LIN {X 0,Y 351.6,Z 693.303,A -85,B 0,C 180,E1 16687.079,E2 16687.079} C_VEL
LIN {X 0,Y 338.557,Z 672.287,A -85,B 0,C 180,E1 16684.342,E2 16684.342} C_VEL
LIN {X 0,Y 333.384,Z 663.984,A -85,B 0,C 180,E1 16683.188,E2 16683.188} C_VEL
LIN {X 0,Y 331.512,Z 660.817,A -85,B 0,C 180,E1 16682.749,E2 16682.749} C_VEL
LIN {X 0,Y 331.209,Z 659.403,A -85,B 0,C 180,E1 16682.628,E2 16682.628} C_VEL
LIN {X 0,Y 331.206,Z 659.412,A -85,B 0,C 180,E1 16678.295,E2 16678.295} C_VEL
LIN {X 0,Y 331.179,Z 659.421,A -85,B 0,C 180,E1 16674.056,E2 16674.056} C_VEL
LIN {X 0,Y 331.185,Z 659.414,A -85,B 0,C 180,E1 16669.63,E2 16669.63} C_VEL
LIN {X 0,Y 331.203,Z 659.41,A -85,B 0,C 180,E1 16665.23,E2 16665.23} C_VEL
LIN {X 0,Y 331.214,Z 659.412,A -85,B 0,C 180,E1 16660.966,E2 16660.966} C_VEL
LIN {X 0,Y 331.187,Z 659.409,A -85,B 0,C 180,E1 16656.686,E2 16656.686} C_VEL
LIN {X 0,Y 331.142,Z 659.398,A -85,B 0,C 180,E1 16652.252,E2 16652.252} C_VEL
LIN {X 0,Y 331.187,Z 659.405,A -85,B 0,C 180,E1 16647.926,E2 16647.926} C_VEL
LIN {X 0,Y 331.208,Z 659.407,A -85,B 0,C 180,E1 16643.589,E2 16643.589} C_VEL
LIN {X 0,Y 331.175,Z 659.386,A -85,B 0,C 180,E1 16639.214,E2 16639.214} C_VEL
LIN {X 0,Y 331.174,Z 659.417,A -85,B 0,C 180,E1 16634.774,E2 16634.774} C_VEL
LIN {X 0,Y 331.205,Z 659.409,A -85,B 0,C 180,E1 16630.36,E2 16630.36} C_VEL
LIN {X 0,Y 331.219,Z 659.406,A -85,B 0,C 180,E1 16626.142,E2 16626.142} C_VEL
LIN {X 0,Y 331.209,Z 659.41,A -85,B 0,C 180,E1 16621.816,E2 16621.816} C_VEL
LIN {X 0,Y 331.153,Z 659.419,A -85,B 0,C 180,E1 16617.493,E2 16617.493} C_VEL
LIN {X 0,Y 331.182,Z 659.552,A -85,B 0,C 180,E1 16615.549,E2 16615.549} C_VEL
LIN {X 0,Y 340.001,Z 685.204,A -85,B 0,C 180,E1 16611.864,E2 16611.864} C_VEL
LIN {X 0,Y 347.057,Z 708.569,A -85,B 0,C 180,E1 16608.722,E2 16608.722} C_VEL
LIN {X 0,Y 350.806,Z 723.326,A -85,B 0,C 180,E1 16606.852,E2 16606.852} C_VEL
LIN {X 0,Y 347.552,Z 765.475,A -85,B 0,C 180,E1 16602.633,E2 16602.633} C_VEL
LIN {X 0,Y 344.201,Z 811.082,A -85,B 0,C 180,E1 16598.076,E2 16598.076} C_VEL
LIN {X 0,Y 341.544,Z 849.928,A -85,B 0,C 180,E1 16594.195,E2 16594.195} C_VEL
LIN {X 0,Y 340.993,Z 853.906,A -85,B 0,C 180,E1 16593.867,E2 16593.867} C_VEL
LIN {X 0,Y 338.603,Z 912.667,A -85,B 0,C 180,E1 16592.158,E2 16592.158} C_VEL
LIN {X 0,Y 337.347,Z 920.247,A -85,B 0,C 180,E1 16591.97,E2 16591.97} C_VEL
LIN {X 0,Y 330.436,Z 940.215,A -85,B 0,C 180,E1 16591.578,E2 16591.578} C_VEL
LIN {X 0,Y 329.472,Z 946.731,A -85,B 0,C 180,E1 16591.405,E2 16591.405} C_VEL
LIN {X 0,Y 328.184,Z 1001.563,A -85,B 0,C 180,E1 16589.68,E2 16589.68} C_VEL
LIN {X 0,Y 327.54,Z 1020.153,A -85,B 0,C 180,E1 16588.728,E2 16588.728} C_VEL
LIN {X 0,Y 326.683,Z 1037.892,A -85,B 0,C 180,E1 16587.432,E2 16587.432} C_VEL
LIN {X 0,Y 325.718,Z 1053.514,A -85,B 0,C 180,E1 16585.921,E2 16585.921} C_VEL
LIN {X 0,Y 324.725,Z 1067.809,A -85,B 0,C 180,E1 16584.171,E2 16584.171} C_VEL
LIN {X 0,Y 323.744,Z 1081.305,A -85,B 0,C 180,E1 16582.105,E2 16582.105} C_VEL
LIN {X 0,Y 322.95,Z 1092.772,A -85,B 0,C 180,E1 16579.907,E2 16579.907} C_VEL
LIN {X 0,Y 322.373,Z 1102.885,A -85,B 0,C 180,E1 16577.505,E2 16577.505} C_VEL
LIN {X 0,Y 322.042,Z 1111.903,A -85,B 0,C 180,E1 16574.745,E2 16574.745} C_VEL
LIN {X 0,Y 322.044,Z 1118.472,A -85,B 0,C 180,E1 16572.052,E2 16572.052} C_VEL
LIN {X 0,Y 322.479,Z 1123.729,A -85,B 0,C 180,E1 16568.915,E2 16568.915} C_VEL
LIN {X 0,Y 323.342,Z 1126.487,A -85,B 0,C 180,E1 16566.031,E2 16566.031} C_VEL
LIN {X 0,Y 324.595,Z 1127.269,A -85,B 0,C 180,E1 16563.351,E2 16563.351} C_VEL
LIN {X 0,Y 326.459,Z 1126.247,A -85,B 0,C 180,E1 16560.523,E2 16560.523} C_VEL
LIN {X 0,Y 328.731,Z 1123.536,A -85,B 0,C 180,E1 16557.905,E2 16557.905} C_VEL
LIN {X 0,Y 331.715,Z 1118.637,A -85,B 0,C 180,E1 16555.155,E2 16555.155} C_VEL
LIN {X 0,Y 335.038,Z 1111.991,A -85,B 0,C 180,E1 16552.623,E2 16552.623} C_VEL
LIN {X 0,Y 338.59,Z 1103.844,A -85,B 0,C 180,E1 16550.306,E2 16550.306} C_VEL
LIN {X 0,Y 342.209,Z 1094.105,A -85,B 0,C 180,E1 16548.195,E2 16548.195} C_VEL
LIN {X 0,Y 345.994,Z 1082.439,A -85,B 0,C 180,E1 16546.204,E2 16546.204} C_VEL
LIN {X 0,Y 349.656,Z 1069.004,A -85,B 0,C 180,E1 16544.403,E2 16544.403} C_VEL
LIN {X 0,Y 352.823,Z 1055.115,A -85,B 0,C 180,E1 16542.94,E2 16542.94} C_VEL
LIN {X 0,Y 355.186,Z 1042.191,A -85,B 0,C 180,E1 16541.873,E2 16541.873} C_VEL
LIN {X 0,Y 357.053,Z 1029.824,A -85,B 0,C 180,E1 16541.04,E2 16541.04} C_VEL
LIN {X 0,Y 358.754,Z 1014.945,A -85,B 0,C 180,E1 16540.256,E2 16540.256} C_VEL
LIN {X 0,Y 361.941,Z 979.464,A -85,B 0,C 180,E1 16538.955,E2 16538.955} C_VEL
LIN {X 0,Y 374.08,Z 877.56,A -85,B 0,C 180,E1 16535.718,E2 16535.718} C_VEL
LIN {X 0,Y 374.117,Z 874.18,A -85,B 0,C 180,E1 16535.44,E2 16535.44} C_VEL
LIN {X 0,Y 384.232,Z 826.781,A -85,B 0,C 180,E1 16530.45,E2 16530.45} C_VEL
LIN {X 0,Y 396.371,Z 779.965,A -85,B 0,C 180,E1 16525.503,E2 16525.503} C_VEL
LIN {X 0,Y 397.772,Z 774.804,A -85,B 0,C 180,E1 16524.94,E2 16524.94} C_VEL
LIN {X 0,Y 397.847,Z 768.846,A -85,B 0,C 180,E1 16523.05,E2 16523.05} C_VEL
LIN {X 0,Y 397.965,Z 764.729,A -85,B 0,C 180,E1 16521.172,E2 16521.172} C_VEL
LIN {X 0,Y 393.008,Z 774.877,A -85,B 0,C 180,E1 16519.215,E2 16519.215} C_VEL
LIN {X 0,Y 388.071,Z 786.864,A -85,B 0,C 180,E1 16518.567,E2 16518.567} C_VEL
LIN {X 0,Y 382.601,Z 800.942,A -85,B 0,C 180,E1 16517.916,E2 16517.916} C_VEL
LIN {X 0,Y 379.821,Z 808.396,A -85,B 0,C 180,E1 16517.481,E2 16517.481} C_VEL
LIN {X 0,Y 375.285,Z 820.645,A -85,B 0,C 180,E1 16516.885,E2 16516.885} C_VEL
LIN {X 0,Y 373.467,Z 826.767,A -85,B 0,C 180,E1 16516.497,E2 16516.497} C_VEL
LIN {X 0,Y 360.759,Z 976.244,A -85,B 0,C 180,E1 16512.41,E2 16512.41} C_VEL
LIN {X 0,Y 357.8,Z 1000.344,A -85,B 0,C 180,E1 16511.472,E2 16511.472} C_VEL
LIN {X 0,Y 354.247,Z 1023.747,A -85,B 0,C 180,E1 16510.265,E2 16510.265} C_VEL
LIN {X 0,Y 350.535,Z 1045.323,A -85,B 0,C 180,E1 16508.852,E2 16508.852} C_VEL
LIN {X 0,Y 346.37,Z 1067.024,A -85,B 0,C 180,E1 16507.106,E2 16507.106} C_VEL
LIN {X 0,Y 342.045,Z 1087.908,A -85,B 0,C 180,E1 16505.059,E2 16505.059} C_VEL
LIN {X 0,Y 337.867,Z 1107.196,A -85,B 0,C 180,E1 16502.787,E2 16502.787} C_VEL
LIN {X 0,Y 333.963,Z 1124.72,A -85,B 0,C 180,E1 16500.333,E2 16500.333} C_VEL
LIN {X 0,Y 330.316,Z 1141.142,A -85,B 0,C 180,E1 16497.587,E2 16497.587} C_VEL
LIN {X 0,Y 327.252,Z 1155.552,A -85,B 0,C 180,E1 16494.743,E2 16494.743} C_VEL
LIN {X 0,Y 324.684,Z 1168.697,A -85,B 0,C 180,E1 16491.685,E2 16491.685} C_VEL
LIN {X 0,Y 322.698,Z 1180.452,A -85,B 0,C 180,E1 16488.421,E2 16488.421} C_VEL
LIN {X 0,Y 321.385,Z 1190.146,A -85,B 0,C 180,E1 16485.147,E2 16485.147} C_VEL
LIN {X 0,Y 320.607,Z 1198.9,A -85,B 0,C 180,E1 16481.511,E2 16481.511} C_VEL
LIN {X 0,Y 320.369,Z 1205.389,A -85,B 0,C 180,E1 16478.071,E2 16478.071} C_VEL
LIN {X 0,Y 320.383,Z 1209.815,A -85,B 0,C 180,E1 16474.831,E2 16474.831} C_VEL
LIN {X 0,Y 320.415,Z 1212.911,A -85,B 0,C 180,E1 16471.607,E2 16471.607} C_VEL
LIN {X 0,Y 320.319,Z 1214.462,A -85,B 0,C 180,E1 16468.388,E2 16468.388} C_VEL
LIN {X 0,Y 320.125,Z 1214.771,A -85,B 0,C 180,E1 16465.151,E2 16465.151} C_VEL
LIN {X 0,Y 320.101,Z 1213.552,A -85,B 0,C 180,E1 16461.555,E2 16461.555} C_VEL
LIN {X 0,Y 320.61,Z 1210.744,A -85,B 0,C 180,E1 16457.754,E2 16457.754} C_VEL
LIN {X 0,Y 322.079,Z 1205.966,A -85,B 0,C 180,E1 16453.773,E2 16453.773} C_VEL
LIN {X 0,Y 324.889,Z 1199.156,A -85,B 0,C 180,E1 16449.647,E2 16449.647} C_VEL
LIN {X 0,Y 328.956,Z 1190.922,A -85,B 0,C 180,E1 16445.771,E2 16445.771} C_VEL
LIN {X 0,Y 335.049,Z 1179.871,A -85,B 0,C 180,E1 16441.671,E2 16441.671} C_VEL
LIN {X 0,Y 342.588,Z 1167.283,A -85,B 0,C 180,E1 16437.912,E2 16437.912} C_VEL
LIN {X 0,Y 351.822,Z 1152.785,A -85,B 0,C 180,E1 16434.363,E2 16434.363} C_VEL
LIN {X 0,Y 363.35,Z 1135.626,A -85,B 0,C 180,E1 16430.935,E2 16430.935} C_VEL
LIN {X 0,Y 376.213,Z 1117.274,A -85,B 0,C 180,E1 16427.95,E2 16427.95} C_VEL
LIN {X 0,Y 390.249,Z 1097.915,A -85,B 0,C 180,E1 16425.407,E2 16425.407} C_VEL
LIN {X 0,Y 399.921,Z 1084.762,A -85,B 0,C 180,E1 16423.961,E2 16423.961} C_VEL
LIN {X 0,Y 385.937,Z 1102.502,A -85,B 0,C 180,E1 16421.551,E2 16421.551} C_VEL
LIN {X 0,Y 372.691,Z 1119.346,A -85,B 0,C 180,E1 16418.694,E2 16418.694} C_VEL
LIN {X 0,Y 361.071,Z 1134.237,A -85,B 0,C 180,E1 16415.562,E2 16415.562} C_VEL
LIN {X 0,Y 351.032,Z 1147.199,A -85,B 0,C 180,E1 16412.189,E2 16412.189} C_VEL
LIN {X 0,Y 342.197,Z 1158.696,A -85,B 0,C 180,E1 16408.446,E2 16408.446} C_VEL
LIN {X 0,Y 335.286,Z 1167.815,A -85,B 0,C 180,E1 16404.681,E2 16404.681} C_VEL
LIN {X 0,Y 330.062,Z 1174.865,A -85,B 0,C 180,E1 16400.948,E2 16400.948} C_VEL
LIN {X 0,Y 325.955,Z 1180.366,A -85,B 0,C 180,E1 16396.947,E2 16396.947} C_VEL
LIN {X 0,Y 323.237,Z 1183.951,A -85,B 0,C 180,E1 16393.054,E2 16393.054} C_VEL
LIN {X 0,Y 321.548,Z 1185.952,A -85,B 0,C 180,E1 16389.129,E2 16389.129} C_VEL
LIN {X 0,Y 320.679,Z 1186.308,A -85,B 0,C 180,E1 16385.371,E2 16385.371} C_VEL
LIN {X 0,Y 320.312,Z 1185.132,A -85,B 0,C 180,E1 16381.793,E2 16381.793} C_VEL
LIN {X 0,Y 320.188,Z 1182.586,A -85,B 0,C 180,E1 16378.214,E2 16378.214} C_VEL
LIN {X 0,Y 320.238,Z 1178.622,A -85,B 0,C 180,E1 16374.809,E2 16374.809} C_VEL
LIN {X 0,Y 320.546,Z 1172.903,A -85,B 0,C 180,E1 16371.212,E2 16371.212} C_VEL
LIN {X 0,Y 321.275,Z 1165.446,A -85,B 0,C 180,E1 16367.604,E2 16367.604} C_VEL
LIN {X 0,Y 322.507,Z 1156.431,A -85,B 0,C 180,E1 16364.171,E2 16364.171} C_VEL
LIN {X 0,Y 324.38,Z 1145.515,A -85,B 0,C 180,E1 16360.746,E2 16360.746} C_VEL
LIN {X 0,Y 326.834,Z 1133.136,A -85,B 0,C 180,E1 16357.509,E2 16357.509} C_VEL
LIN {X 0,Y 329.765,Z 1119.49,A -85,B 0,C 180,E1 16354.501,E2 16354.501} C_VEL
LIN {X 0,Y 333.361,Z 1103.336,A -85,B 0,C 180,E1 16351.521,E2 16351.521} C_VEL
LIN {X 0,Y 337.081,Z 1086.696,A -85,B 0,C 180,E1 16348.931,E2 16348.931} C_VEL
LIN {X 0,Y 341.193,Z 1067.985,A -85,B 0,C 180,E1 16346.473,E2 16346.473} C_VEL
LIN {X 0,Y 345.292,Z 1048.376,A -85,B 0,C 180,E1 16344.308,E2 16344.308} C_VEL
LIN {X 0,Y 349.263,Z 1028.055,A -85,B 0,C 180,E1 16342.431,E2 16342.431} C_VEL
LIN {X 0,Y 353.169,Z 1005.858,A -85,B 0,C 180,E1 16340.751,E2 16340.751} C_VEL
LIN {X 0,Y 356.624,Z 983.295,A -85,B 0,C 180,E1 16339.375,E2 16339.375} C_VEL
LIN {X 0,Y 359.63,Z 960.074,A -85,B 0,C 180,E1 16338.262,E2 16338.262} C_VEL
LIN {X 0,Y 362.141,Z 935.797,A -85,B 0,C 180,E1 16337.391,E2 16337.391} C_VEL
LIN {X 0,Y 377.659,Z 753.869,A -85,B 0,C 180,E1 16332.538,E2 16332.538} C_VEL
LIN {X 0,Y 361.552,Z 724.578,A -85,B 0,C 180,E1 16329.605,E2 16329.605} C_VEL
LIN {X 0,Y 345.257,Z 696.732,A -85,B 0,C 180,E1 16326.37,E2 16326.37} C_VEL
LIN {X 0,Y 331.073,Z 673.869,A -85,B 0,C 180,E1 16323.295,E2 16323.295} C_VEL
LIN {X 0,Y 326.253,Z 665.854,A -85,B 0,C 180,E1 16322.151,E2 16322.151} C_VEL
LIN {X 0,Y 323.79,Z 662.4,A -85,B 0,C 180,E1 16321.583,E2 16321.583} C_VEL
LIN {X 0,Y 323.27,Z 660.399,A -85,B 0,C 180,E1 16321.395,E2 16321.395} C_VEL
LIN {X 0,Y 323.265,Z 660.4,A -85,B 0,C 180,E1 16317.036,E2 16317.036} C_VEL
LIN {X 0,Y 323.21,Z 660.4,A -85,B 0,C 180,E1 16312.752,E2 16312.752} C_VEL
LIN {X 0,Y 323.236,Z 660.391,A -85,B 0,C 180,E1 16308.208,E2 16308.208} C_VEL
LIN {X 0,Y 323.28,Z 660.382,A -85,B 0,C 180,E1 16303.963,E2 16303.963} C_VEL
LIN {X 0,Y 323.26,Z 660.392,A -85,B 0,C 180,E1 16299.617,E2 16299.617} C_VEL
LIN {X 0,Y 323.239,Z 660.407,A -85,B 0,C 180,E1 16295.327,E2 16295.327} C_VEL
LIN {X 0,Y 323.238,Z 660.398,A -85,B 0,C 180,E1 16290.711,E2 16290.711} C_VEL
LIN {X 0,Y 323.258,Z 660.376,A -85,B 0,C 180,E1 16286.456,E2 16286.456} C_VEL
LIN {X 0,Y 323.277,Z 660.401,A -85,B 0,C 180,E1 16282.181,E2 16282.181} C_VEL
LIN {X 0,Y 323.219,Z 660.38,A -85,B 0,C 180,E1 16277.814,E2 16277.814} C_VEL
LIN {X 0,Y 323.22,Z 660.402,A -85,B 0,C 180,E1 16273.283,E2 16273.283} C_VEL
LIN {X 0,Y 323.275,Z 660.397,A -85,B 0,C 180,E1 16268.977,E2 16268.977} C_VEL
LIN {X 0,Y 323.27,Z 660.398,A -85,B 0,C 180,E1 16264.54,E2 16264.54} C_VEL
LIN {X 0,Y 323.266,Z 660.401,A -85,B 0,C 180,E1 16260.136,E2 16260.136} C_VEL
LIN {X 0,Y 323.262,Z 660.562,A -85,B 0,C 180,E1 16256.23,E2 16256.23} C_VEL
LIN {X 0,Y 332.107,Z 686.213,A -85,B 0,C 180,E1 16252.438,E2 16252.438} C_VEL
LIN {X 0,Y 339.096,Z 708.964,A -85,B 0,C 180,E1 16249.337,E2 16249.337} C_VEL
LIN {X 0,Y 343.3,Z 725.338,A -85,B 0,C 180,E1 16247.214,E2 16247.214} C_VEL
LIN {X 0,Y 339.888,Z 767.707,A -85,B 0,C 180,E1 16242.907,E2 16242.907} C_VEL
LIN {X 0,Y 336.445,Z 813.005,A -85,B 0,C 180,E1 16238.322,E2 16238.322} C_VEL
LIN {X 0,Y 333.814,Z 850.452,A -85,B 0,C 180,E1 16234.547,E2 16234.547} C_VEL
LIN {X 0,Y 333.202,Z 854.884,A -85,B 0,C 180,E1 16234.176,E2 16234.176} C_VEL
LIN {X 0,Y 329.472,Z 946.731,A -85,B 0,C 180,E1 16231.405,E2 16231.405} C_VEL
LIN {X 0,Y 328.234,Z 954.316,A -85,B 0,C 180,E1 16231.213,E2 16231.213} C_VEL
LIN {X 0,Y 321.52,Z 974.314,A -85,B 0,C 180,E1 16230.785,E2 16230.785} C_VEL
LIN {X 0,Y 320.651,Z 980.824,A -85,B 0,C 180,E1 16230.599,E2 16230.599} C_VEL
LIN {X 0,Y 320.189,Z 1004.569,A -85,B 0,C 180,E1 16229.757,E2 16229.757} C_VEL
LIN {X 0,Y 319.534,Z 1022.035,A -85,B 0,C 180,E1 16228.804,E2 16228.804} C_VEL
LIN {X 0,Y 318.651,Z 1039.614,A -85,B 0,C 180,E1 16227.464,E2 16227.464} C_VEL
LIN {X 0,Y 317.568,Z 1056.514,A -85,B 0,C 180,E1 16225.749,E2 16225.749} C_VEL
LIN {X 0,Y 316.523,Z 1071.125,A -85,B 0,C 180,E1 16223.846,E2 16223.846} C_VEL
LIN {X 0,Y 315.618,Z 1083.502,A -85,B 0,C 180,E1 16221.848,E2 16221.848} C_VEL
LIN {X 0,Y 314.818,Z 1095.345,A -85,B 0,C 180,E1 16219.476,E2 16219.476} C_VEL
LIN {X 0,Y 314.289,Z 1105.102,A -85,B 0,C 180,E1 16217.015,E2 16217.015} C_VEL
LIN {X 0,Y 314.038,Z 1112.827,A -85,B 0,C 180,E1 16214.564,E2 16214.564} C_VEL
LIN {X 0,Y 314.064,Z 1119.146,A -85,B 0,C 180,E1 16211.939,E2 16211.939} C_VEL
LIN {X 0,Y 314.491,Z 1124.273,A -85,B 0,C 180,E1 16208.958,E2 16208.958} C_VEL
LIN {X 0,Y 315.309,Z 1127.161,A -85,B 0,C 180,E1 16206.186,E2 16206.186} C_VEL
LIN {X 0,Y 316.69,Z 1128.397,A -85,B 0,C 180,E1 16203.254,E2 16203.254} C_VEL
LIN {X 0,Y 318.499,Z 1127.771,A -85,B 0,C 180,E1 16200.536,E2 16200.536} C_VEL
LIN {X 0,Y 321.014,Z 1125.248,A -85,B 0,C 180,E1 16197.676,E2 16197.676} C_VEL
LIN {X 0,Y 323.921,Z 1121.033,A -85,B 0,C 180,E1 16195.038,E2 16195.038} C_VEL
LIN {X 0,Y 327.377,Z 1114.938,A -85,B 0,C 180,E1 16192.45,E2 16192.45} C_VEL
LIN {X 0,Y 331.048,Z 1107.261,A -85,B 0,C 180,E1 16190.083,E2 16190.083} C_VEL
LIN {X 0,Y 335.132,Z 1097.416,A -85,B 0,C 180,E1 16187.767,E2 16187.767} C_VEL
LIN {X 0,Y 339.254,Z 1085.775,A -85,B 0,C 180,E1 16185.663,E2 16185.663} C_VEL
LIN {X 0,Y 342.952,Z 1073.599,A -85,B 0,C 180,E1 16183.917,E2 16183.917} C_VEL
LIN {X 0,Y 346.646,Z 1059.102,A -85,B 0,C 180,E1 16182.28,E2 16182.28} C_VEL
LIN {X 0,Y 349.513,Z 1044.986,A -85,B 0,C 180,E1 16181.049,E2 16181.049} C_VEL
LIN {X 0,Y 351.668,Z 1031.799,A -85,B 0,C 180,E1 16180.134,E2 16180.134} C_VEL
LIN {X 0,Y 353.549,Z 1016.864,A -85,B 0,C 180,E1 16179.321,E2 16179.321} C_VEL
LIN {X 0,Y 356.91,Z 982.076,A -85,B 0,C 180,E1 16178.009,E2 16178.009} C_VEL
LIN {X 0,Y 369.793,Z 879.555,A -85,B 0,C 180,E1 16174.706,E2 16174.706} C_VEL
LIN {X 0,Y 369.885,Z 875.582,A -85,B 0,C 180,E1 16174.369,E2 16174.369} C_VEL
LIN {X 0,Y 380.72,Z 828.557,A -85,B 0,C 180,E1 16169.366,E2 16169.366} C_VEL
LIN {X 0,Y 393.638,Z 782.212,A -85,B 0,C 180,E1 16164.428,E2 16164.428} C_VEL
LIN {X 0,Y 394.254,Z 780.161,A -85,B 0,C 180,E1 16164.183,E2 16164.183} C_VEL
LIN {X 0,Y 394.516,Z 775.16,A -85,B 0,C 180,E1 16162.489,E2 16162.489} C_VEL
LIN {X 0,Y 394.594,Z 772.929,A -85,B 0,C 180,E1 16161.435,E2 16161.435} C_VEL
LIN {X 0,Y 391.433,Z 779.006,A -85,B 0,C 180,E1 16160.25,E2 16160.25} C_VEL
LIN {X 0,Y 386.062,Z 791.611,A -85,B 0,C 180,E1 16159.588,E2 16159.588} C_VEL
LIN {X 0,Y 380.91,Z 804.167,A -85,B 0,C 180,E1 16158.994,E2 16158.994} C_VEL
LIN {X 0,Y 378.371,Z 810.59,A -85,B 0,C 180,E1 16158.63,E2 16158.63} C_VEL
LIN {X 0,Y 373.759,Z 822.721,A -85,B 0,C 180,E1 16158.044,E2 16158.044} C_VEL
LIN {X 0,Y 371.395,Z 829.195,A -85,B 0,C 180,E1 16157.644,E2 16157.644} C_VEL
LIN {X 0,Y 366.908,Z 841.382,A -85,B 0,C 180,E1 16157.052,E2 16157.052} C_VEL
LIN {X 0,Y 364.736,Z 848.726,A -85,B 0,C 180,E1 16156.579,E2 16156.579} C_VEL
LIN {X 0,Y 353.63,Z 976.176,A -85,B 0,C 180,E1 16152.993,E2 16152.993} C_VEL
LIN {X 0,Y 350.574,Z 1000.358,A -85,B 0,C 180,E1 16152.028,E2 16152.028} C_VEL
LIN {X 0,Y 346.842,Z 1024.248,A -85,B 0,C 180,E1 16150.762,E2 16150.762} C_VEL
LIN {X 0,Y 342.882,Z 1046.55,A -85,B 0,C 180,E1 16149.253,E2 16149.253} C_VEL
LIN {X 0,Y 338.623,Z 1068.048,A -85,B 0,C 180,E1 16147.461,E2 16147.461} C_VEL
LIN {X 0,Y 334.225,Z 1088.709,A -85,B 0,C 180,E1 16145.369,E2 16145.369} C_VEL
LIN {X 0,Y 329.981,Z 1107.78,A -85,B 0,C 180,E1 16143.05,E2 16143.05} C_VEL
LIN {X 0,Y 325.97,Z 1125.401,A -85,B 0,C 180,E1 16140.505,E2 16140.505} C_VEL
LIN {X 0,Y 322.1,Z 1142.524,A -85,B 0,C 180,E1 16137.548,E2 16137.548} C_VEL
LIN {X 0,Y 318.872,Z 1157.497,A -85,B 0,C 180,E1 16134.448,E2 16134.448} C_VEL
LIN {X 0,Y 316.368,Z 1170.254,A -85,B 0,C 180,E1 16131.31,E2 16131.31} C_VEL
LIN {X 0,Y 314.464,Z 1181.679,A -85,B 0,C 180,E1 16127.962,E2 16127.962} C_VEL
LIN {X 0,Y 313.19,Z 1191.644,A -85,B 0,C 180,E1 16124.417,E2 16124.417} C_VEL
LIN {X 0,Y 312.563,Z 1199.553,A -85,B 0,C 180,E1 16120.877,E2 16120.877} C_VEL
LIN {X 0,Y 312.392,Z 1205.985,A -85,B 0,C 180,E1 16117.168,E2 16117.168} C_VEL
LIN {X 0,Y 312.434,Z 1209.957,A -85,B 0,C 180,E1 16114.035,E2 16114.035} C_VEL
LIN {X 0,Y 312.435,Z 1212.839,A -85,B 0,C 180,E1 16110.548,E2 16110.548} C_VEL
LIN {X 0,Y 312.282,Z 1214.096,A -85,B 0,C 180,E1 16107.428,E2 16107.428} C_VEL
LIN {X 0,Y 312.088,Z 1214.103,A -85,B 0,C 180,E1 16103.744,E2 16103.744} C_VEL
LIN {X 0,Y 312.21,Z 1212.529,A -85,B 0,C 180,E1 16100.039,E2 16100.039} C_VEL
LIN {X 0,Y 313.125,Z 1209.115,A -85,B 0,C 180,E1 16095.952,E2 16095.952} C_VEL
LIN {X 0,Y 315.156,Z 1204.057,A -85,B 0,C 180,E1 16091.883,E2 16091.883} C_VEL
LIN {X 0,Y 318.684,Z 1196.848,A -85,B 0,C 180,E1 16087.686,E2 16087.686} C_VEL
LIN {X 0,Y 323.861,Z 1187.722,A -85,B 0,C 180,E1 16083.559,E2 16083.559} C_VEL
LIN {X 0,Y 330.932,Z 1176.45,A -85,B 0,C 180,E1 16079.494,E2 16079.494} C_VEL
LIN {X 0,Y 339.949,Z 1163.132,A -85,B 0,C 180,E1 16075.614,E2 16075.614} C_VEL
LIN {X 0,Y 350.881,Z 1147.859,A -85,B 0,C 180,E1 16072.008,E2 16072.008} C_VEL
LIN {X 0,Y 363.738,Z 1130.623,A -85,B 0,C 180,E1 16068.718,E2 16068.718} C_VEL
LIN {X 0,Y 377.904,Z 1112.389,A -85,B 0,C 180,E1 16065.902,E2 16065.902} C_VEL
LIN {X 0,Y 390.605,Z 1096.484,A -85,B 0,C 180,E1 16063.878,E2 16063.878} C_VEL
LIN {X 0,Y 375.998,Z 1113.412,A -85,B 0,C 180,E1 16061.265,E2 16061.265} C_VEL
LIN {X 0,Y 362.862,Z 1128.688,A -85,B 0,C 180,E1 16058.32,E2 16058.32} C_VEL
LIN {X 0,Y 351.359,Z 1142.172,A -85,B 0,C 180,E1 16055.092,E2 16055.092} C_VEL
LIN {X 0,Y 341.04,Z 1154.34,A -85,B 0,C 180,E1 16051.462,E2 16051.462} C_VEL
LIN {X 0,Y 332.446,Z 1164.563,A -85,B 0,C 180,E1 16047.596,E2 16047.596} C_VEL
LIN {X 0,Y 325.527,Z 1172.862,A -85,B 0,C 180,E1 16043.539,E2 16043.539} C_VEL
LIN {X 0,Y 320.433,Z 1179.04,A -85,B 0,C 180,E1 16039.509,E2 16039.509} C_VEL
LIN {X 0,Y 316.617,Z 1183.591,A -85,B 0,C 180,E1 16035.199,E2 16035.199} C_VEL
LIN {X 0,Y 314.252,Z 1186.098,A -85,B 0,C 180,E1 16031.01,E2 16031.01} C_VEL
LIN {X 0,Y 312.984,Z 1186.858,A -85,B 0,C 180,E1 16026.977,E2 16026.977} C_VEL
LIN {X 0,Y 312.435,Z 1186.167,A -85,B 0,C 180,E1 16023.306,E2 16023.306} C_VEL
LIN {X 0,Y 312.22,Z 1183.908,A -85,B 0,C 180,E1 16019.637,E2 16019.637} C_VEL
LIN {X 0,Y 312.198,Z 1180.222,A -85,B 0,C 180,E1 16015.964,E2 16015.964} C_VEL
LIN {X 0,Y 312.402,Z 1175.198,A -85,B 0,C 180,E1 16012.464,E2 16012.464} C_VEL
LIN {X 0,Y 312.988,Z 1168.178,A -85,B 0,C 180,E1 16008.767,E2 16008.767} C_VEL
LIN {X 0,Y 314.041,Z 1159.797,A -85,B 0,C 180,E1 16005.248,E2 16005.248} C_VEL
LIN {X 0,Y 315.727,Z 1149.522,A -85,B 0,C 180,E1 16001.733,E2 16001.733} C_VEL
LIN {X 0,Y 317.991,Z 1137.772,A -85,B 0,C 180,E1 15998.419,E2 15998.419} C_VEL
LIN {X 0,Y 320.957,Z 1123.886,A -85,B 0,C 180,E1 15995.134,E2 15995.134} C_VEL
LIN {X 0,Y 324.445,Z 1108.467,A -85,B 0,C 180,E1 15992.072,E2 15992.072} C_VEL
LIN {X 0,Y 328.359,Z 1091.5,A -85,B 0,C 180,E1 15989.236,E2 15989.236} C_VEL
LIN {X 0,Y 332.575,Z 1072.887,A -85,B 0,C 180,E1 15986.625,E2 15986.625} C_VEL
LIN {X 0,Y 336.846,Z 1053.182,A -85,B 0,C 180,E1 15984.323,E2 15984.323} C_VEL
LIN {X 0,Y 340.989,Z 1032.596,A -85,B 0,C 180,E1 15982.316,E2 15982.316} C_VEL
LIN {X 0,Y 344.936,Z 1011.293,A -85,B 0,C 180,E1 15980.598,E2 15980.598} C_VEL
LIN {X 0,Y 348.736,Z 987.99,A -85,B 0,C 180,E1 15979.075,E2 15979.075} C_VEL
LIN {X 0,Y 351.96,Z 964.592,A -85,B 0,C 180,E1 15977.868,E2 15977.868} C_VEL
LIN {X 0,Y 354.625,Z 941.038,A -85,B 0,C 180,E1 15976.948,E2 15976.948} C_VEL
LIN {X 0,Y 370.957,Z 756.717,A -85,B 0,C 180,E1 15971.904,E2 15971.904} C_VEL
LIN {X 0,Y 355.167,Z 728.093,A -85,B 0,C 180,E1 15968.968,E2 15968.968} C_VEL
LIN {X 0,Y 339.851,Z 701.768,A -85,B 0,C 180,E1 15965.84,E2 15965.84} C_VEL
LIN {X 0,Y 325.976,Z 679.24,A -85,B 0,C 180,E1 15962.755,E2 15962.755} C_VEL
LIN {X 0,Y 320.176,Z 670.203,A -85,B 0,C 180,E1 15961.385,E2 15961.385} C_VEL
LIN {X 0,Y 317.637,Z 666.073,A -85,B 0,C 180,E1 15960.763,E2 15960.763} C_VEL
LIN {X 0,Y 315.671,Z 662.88,A -85,B 0,C 180,E1 15960.269,E2 15960.269} C_VEL
LIN {X 0,Y 315.338,Z 661.384,A -85,B 0,C 180,E1 15960.121,E2 15960.121} C_VEL
LIN {X 0,Y 315.325,Z 661.383,A -85,B 0,C 180,E1 15955.751,E2 15955.751} C_VEL
LIN {X 0,Y 315.293,Z 661.388,A -85,B 0,C 180,E1 15951.391,E2 15951.391} C_VEL
LIN {X 0,Y 315.307,Z 661.386,A -85,B 0,C 180,E1 15946.965,E2 15946.965} C_VEL
LIN {X 0,Y 315.331,Z 661.378,A -85,B 0,C 180,E1 15942.431,E2 15942.431} C_VEL
LIN {X 0,Y 315.304,Z 661.374,A -85,B 0,C 180,E1 15938.023,E2 15938.023} C_VEL
LIN {X 0,Y 315.27,Z 661.381,A -85,B 0,C 180,E1 15933.639,E2 15933.639} C_VEL
LIN {X 0,Y 315.334,Z 661.389,A -85,B 0,C 180,E1 15929.094,E2 15929.094} C_VEL
LIN {X 0,Y 315.332,Z 661.374,A -85,B 0,C 180,E1 15924.544,E2 15924.544} C_VEL
LIN {X 0,Y 315.324,Z 661.371,A -85,B 0,C 180,E1 15920.328,E2 15920.328} C_VEL
LIN {X 0,Y 315.268,Z 661.395,A -85,B 0,C 180,E1 15915.868,E2 15915.868} C_VEL
LIN {X 0,Y 315.305,Z 661.392,A -85,B 0,C 180,E1 15911.323,E2 15911.323} C_VEL
LIN {X 0,Y 315.341,Z 661.384,A -85,B 0,C 180,E1 15907.048,E2 15907.048} C_VEL
LIN {X 0,Y 315.32,Z 661.391,A -85,B 0,C 180,E1 15902.598,E2 15902.598} C_VEL
LIN {X 0,Y 315.299,Z 661.393,A -85,B 0,C 180,E1 15898.191,E2 15898.191} C_VEL
LIN {X 0,Y 315.292,Z 661.56,A -85,B 0,C 180,E1 15896.92,E2 15896.92} C_VEL
LIN {X 0,Y 323.499,Z 684.986,A -85,B 0,C 180,E1 15893.382,E2 15893.382} C_VEL
LIN {X 0,Y 330.553,Z 707.56,A -85,B 0,C 180,E1 15890.196,E2 15890.196} C_VEL
LIN {X 0,Y 335.832,Z 726.986,A -85,B 0,C 180,E1 15887.626,E2 15887.626} C_VEL
LIN {X 0,Y 332.262,Z 769.966,A -85,B 0,C 180,E1 15883.206,E2 15883.206} C_VEL
LIN {X 0,Y 328.695,Z 815.01,A -85,B 0,C 180,E1 15878.574,E2 15878.574} C_VEL
LIN {X 0,Y 326.04,Z 851.112,A -85,B 0,C 180,E1 15874.881,E2 15874.881} C_VEL
LIN {X 0,Y 325.416,Z 855.577,A -85,B 0,C 180,E1 15874.497,E2 15874.497} C_VEL
LIN {X 0,Y 320.651,Z 980.824,A -85,B 0,C 180,E1 15870.599,E2 15870.599} C_VEL
LIN {X 0,Y 319.501,Z 988.411,A -85,B 0,C 180,E1 15870.385,E2 15870.385} C_VEL
LIN {X 0,Y 313.092,Z 1007.242,A -85,B 0,C 180,E1 15869.808,E2 15869.808} C_VEL
LIN {X 0,Y 311.917,Z 1014.671,A -85,B 0,C 180,E1 15869.444,E2 15869.444} C_VEL
LIN {X 0,Y 311.141,Z 1031.69,A -85,B 0,C 180,E1 15868.3,E2 15868.3} C_VEL
LIN {X 0,Y 310.24,Z 1047.214,A -85,B 0,C 180,E1 15866.92,E2 15866.92} C_VEL
LIN {X 0,Y 309.148,Z 1063.124,A -85,B 0,C 180,E1 15865.102,E2 15865.102} C_VEL
LIN {X 0,Y 308.096,Z 1077.46,A -85,B 0,C 180,E1 15863.016,E2 15863.016} C_VEL
LIN {X 0,Y 307.259,Z 1088.961,A -85,B 0,C 180,E1 15860.949,E2 15860.949} C_VEL
LIN {X 0,Y 306.537,Z 1100.542,A -85,B 0,C 180,E1 15858.35,E2 15858.35} C_VEL
LIN {X 0,Y 306.127,Z 1109.715,A -85,B 0,C 180,E1 15855.725,E2 15855.725} C_VEL
LIN {X 0,Y 306.024,Z 1117.129,A -85,B 0,C 180,E1 15853.025,E2 15853.025} C_VEL
LIN {X 0,Y 306.248,Z 1122.552,A -85,B 0,C 180,E1 15850.341,E2 15850.341} C_VEL
LIN {X 0,Y 306.888,Z 1126.665,A -85,B 0,C 180,E1 15847.484,E2 15847.484} C_VEL
LIN {X 0,Y 307.987,Z 1128.93,A -85,B 0,C 180,E1 15844.651,E2 15844.651} C_VEL
LIN {X 0,Y 309.719,Z 1129.496,A -85,B 0,C 180,E1 15841.661,E2 15841.661} C_VEL
LIN {X 0,Y 311.902,Z 1128.278,A -85,B 0,C 180,E1 15838.894,E2 15838.894} C_VEL
LIN {X 0,Y 314.85,Z 1125.099,A -85,B 0,C 180,E1 15835.99,E2 15835.99} C_VEL
LIN {X 0,Y 318.204,Z 1120.259,A -85,B 0,C 180,E1 15833.32,E2 15833.32} C_VEL
LIN {X 0,Y 322.376,Z 1112.876,A -85,B 0,C 180,E1 15830.535,E2 15830.535} C_VEL
LIN {X 0,Y 326.491,Z 1104.274,A -85,B 0,C 180,E1 15828.156,E2 15828.156} C_VEL
LIN {X 0,Y 330.706,Z 1094.214,A -85,B 0,C 180,E1 15825.999,E2 15825.999} C_VEL
LIN {X 0,Y 335.212,Z 1081.515,A -85,B 0,C 180,E1 15823.891,E2 15823.891} C_VEL
LIN {X 0,Y 339.021,Z 1068.722,A -85,B 0,C 180,E1 15822.223,E2 15822.223} C_VEL
LIN {X 0,Y 342.624,Z 1054.348,A -85,B 0,C 180,E1 15820.742,E2 15820.742} C_VEL
LIN {X 0,Y 345.894,Z 1037.75,A -85,B 0,C 180,E1 15819.434,E2 15819.434} C_VEL
LIN {X 0,Y 348.428,Z 1020.013,A -85,B 0,C 180,E1 15818.402,E2 15818.402} C_VEL
LIN {X 0,Y 351.701,Z 988.068,A -85,B 0,C 180,E1 15817.14,E2 15817.14} C_VEL
LIN {X 0,Y 365.822,Z 881.597,A -85,B 0,C 180,E1 15813.652,E2 15813.652} C_VEL
LIN {X 0,Y 365.9,Z 877.258,A -85,B 0,C 180,E1 15813.284,E2 15813.284} C_VEL
LIN {X 0,Y 377.653,Z 829.877,A -85,B 0,C 180,E1 15808.195,E2 15808.195} C_VEL
LIN {X 0,Y 390.803,Z 785.711,A -85,B 0,C 180,E1 15803.45,E2 15803.45} C_VEL
LIN {X 0,Y 391.283,Z 781.073,A -85,B 0,C 180,E1 15801.721,E2 15801.721} C_VEL
LIN {X 0,Y 389.941,Z 783.573,A -85,B 0,C 180,E1 15801.266,E2 15801.266} C_VEL
LIN {X 0,Y 385.324,Z 793.928,A -85,B 0,C 180,E1 15800.725,E2 15800.725} C_VEL
LIN {X 0,Y 379.787,Z 806.767,A -85,B 0,C 180,E1 15800.121,E2 15800.121} C_VEL
LIN {X 0,Y 377.139,Z 813.174,A -85,B 0,C 180,E1 15799.775,E2 15799.775} C_VEL
LIN {X 0,Y 372.045,Z 825.762,A -85,B 0,C 180,E1 15799.156,E2 15799.156} C_VEL
LIN {X 0,Y 369.935,Z 831.172,A -85,B 0,C 180,E1 15798.825,E2 15798.825} C_VEL
LIN {X 0,Y 365.3,Z 843.548,A -85,B 0,C 180,E1 15798.23,E2 15798.23} C_VEL
LIN {X 0,Y 362.631,Z 850.994,A -85,B 0,C 180,E1 15797.756,E2 15797.756} C_VEL
LIN {X 0,Y 358.094,Z 863.554,A -85,B 0,C 180,E1 15797.131,E2 15797.131} C_VEL
LIN {X 0,Y 355.895,Z 871.125,A -85,B 0,C 180,E1 15796.635,E2 15796.635} C_VEL
LIN {X 0,Y 346.5,Z 976.009,A -85,B 0,C 180,E1 15793.587,E2 15793.587} C_VEL
LIN {X 0,Y 343.385,Z 1000.066,A -85,B 0,C 180,E1 15792.606,E2 15792.606} C_VEL
LIN {X 0,Y 339.647,Z 1023.45,A -85,B 0,C 180,E1 15791.345,E2 15791.345} C_VEL
LIN {X 0,Y 335.632,Z 1045.612,A -85,B 0,C 180,E1 15789.826,E2 15789.826} C_VEL
LIN {X 0,Y 331.271,Z 1067.19,A -85,B 0,C 180,E1 15788.002,E2 15788.002} C_VEL
LIN {X 0,Y 326.59,Z 1088.662,A -85,B 0,C 180,E1 15785.783,E2 15785.783} C_VEL
LIN {X 0,Y 322.102,Z 1108.309,A -85,B 0,C 180,E1 15783.326,E2 15783.326} C_VEL
LIN {X 0,Y 318.032,Z 1125.784,A -85,B 0,C 180,E1 15780.72,E2 15780.72} C_VEL
LIN {X 0,Y 314.21,Z 1142.341,A -85,B 0,C 180,E1 15777.784,E2 15777.784} C_VEL
LIN {X 0,Y 311.007,Z 1156.864,A -85,B 0,C 180,E1 15774.702,E2 15774.702} C_VEL
LIN {X 0,Y 308.442,Z 1169.659,A -85,B 0,C 180,E1 15771.486,E2 15771.486} C_VEL
LIN {X 0,Y 306.497,Z 1181.133,A -85,B 0,C 180,E1 15768.051,E2 15768.051} C_VEL
LIN {X 0,Y 305.258,Z 1190.624,A -85,B 0,C 180,E1 15764.606,E2 15764.606} C_VEL
LIN {X 0,Y 304.602,Z 1198.664,A -85,B 0,C 180,E1 15760.973,E2 15760.973} C_VEL
LIN {X 0,Y 304.422,Z 1204.948,A -85,B 0,C 180,E1 15757.357,E2 15757.357} C_VEL
LIN {X 0,Y 304.468,Z 1209.037,A -85,B 0,C 180,E1 15754.141,E2 15754.141} C_VEL
LIN {X 0,Y 304.471,Z 1212.026,A -85,B 0,C 180,E1 15750.75,E2 15750.75} C_VEL
LIN {X 0,Y 304.301,Z 1213.484,A -85,B 0,C 180,E1 15747.361,E2 15747.361} C_VEL
LIN {X 0,Y 304.099,Z 1213.713,A -85,B 0,C 180,E1 15743.768,E2 15743.768} C_VEL
LIN {X 0,Y 304.239,Z 1212.248,A -85,B 0,C 180,E1 15739.775,E2 15739.775} C_VEL
LIN {X 0,Y 305.244,Z 1209.089,A -85,B 0,C 180,E1 15735.582,E2 15735.582} C_VEL
LIN {X 0,Y 307.432,Z 1204.209,A -85,B 0,C 180,E1 15731.411,E2 15731.411} C_VEL
LIN {X 0,Y 311.199,Z 1197.33,A -85,B 0,C 180,E1 15727.119,E2 15727.119} C_VEL
LIN {X 0,Y 316.906,Z 1188.283,A -85,B 0,C 180,E1 15722.772,E2 15722.772} C_VEL
LIN {X 0,Y 324.555,Z 1177.264,A -85,B 0,C 180,E1 15718.587,E2 15718.587} C_VEL
LIN {X 0,Y 334.445,Z 1163.922,A -85,B 0,C 180,E1 15714.547,E2 15714.547} C_VEL
LIN {X 0,Y 345.97,Z 1149.159,A -85,B 0,C 180,E1 15710.945,E2 15710.945} C_VEL
LIN {X 0,Y 359.459,Z 1132.695,A -85,B 0,C 180,E1 15707.687,E2 15707.687} C_VEL
LIN {X 0,Y 374.213,Z 1115.357,A -85,B 0,C 180,E1 15704.919,E2 15704.919} C_VEL
LIN {X 0,Y 381.323,Z 1107.206,A -85,B 0,C 180,E1 15703.812,E2 15703.812} C_VEL
LIN {X 0,Y 365.997,Z 1123.454,A -85,B 0,C 180,E1 15700.974,E2 15700.974} C_VEL
LIN {X 0,Y 352.462,Z 1137.859,A -85,B 0,C 180,E1 15697.793,E2 15697.793} C_VEL
LIN {X 0,Y 340.684,Z 1150.467,A -85,B 0,C 180,E1 15694.302,E2 15694.302} C_VEL
LIN {X 0,Y 330.658,Z 1161.238,A -85,B 0,C 180,E1 15690.536,E2 15690.536} C_VEL
LIN {X 0,Y 322.377,Z 1170.175,A -85,B 0,C 180,E1 15686.532,E2 15686.532} C_VEL
LIN {X 0,Y 315.581,Z 1177.519,A -85,B 0,C 180,E1 15682.154,E2 15682.154} C_VEL
LIN {X 0,Y 310.917,Z 1182.519,A -85,B 0,C 180,E1 15677.986,E2 15677.986} C_VEL
LIN {X 0,Y 307.593,Z 1185.889,A -85,B 0,C 180,E1 15673.594,E2 15673.594} C_VEL
LIN {X 0,Y 305.672,Z 1187.292,A -85,B 0,C 180,E1 15669.417,E2 15669.417} C_VEL
LIN {X 0,Y 304.678,Z 1187.072,A -85,B 0,C 180,E1 15665.276,E2 15665.276} C_VEL
LIN {X 0,Y 304.306,Z 1185.467,A -85,B 0,C 180,E1 15661.51,E2 15661.51} C_VEL
LIN {X 0,Y 304.185,Z 1182.401,A -85,B 0,C 180,E1 15657.87,E2 15657.87} C_VEL
LIN {X 0,Y 304.273,Z 1177.879,A -85,B 0,C 180,E1 15654.157,E2 15654.157} C_VEL
LIN {X 0,Y 304.639,Z 1171.903,A -85,B 0,C 180,E1 15650.559,E2 15650.559} C_VEL
LIN {X 0,Y 305.5,Z 1163.826,A -85,B 0,C 180,E1 15646.76,E2 15646.76} C_VEL
LIN {X 0,Y 306.928,Z 1154.336,A -85,B 0,C 180,E1 15643.15,E2 15643.15} C_VEL
LIN {X 0,Y 309.072,Z 1142.835,A -85,B 0,C 180,E1 15639.554,E2 15639.554} C_VEL
LIN {X 0,Y 311.825,Z 1129.737,A -85,B 0,C 180,E1 15636.175,E2 15636.175} C_VEL
LIN {X 0,Y 315.112,Z 1115.204,A -85,B 0,C 180,E1 15633.02,E2 15633.02} C_VEL
LIN {X 0,Y 319.1,Z 1098.171,A -85,B 0,C 180,E1 15629.916,E2 15629.916} C_VEL
LIN {X 0,Y 323.216,Z 1080.613,A -85,B 0,C 180,E1 15627.228,E2 15627.228} C_VEL
LIN {X 0,Y 327.551,Z 1061.509,A -85,B 0,C 180,E1 15624.77,E2 15624.77} C_VEL
LIN {X 0,Y 332.018,Z 1040.671,A -85,B 0,C 180,E1 15622.537,E2 15622.537} C_VEL
LIN {X 0,Y 336.32,Z 1018.691,A -85,B 0,C 180,E1 15620.605,E2 15620.605} C_VEL
LIN {X 0,Y 340.125,Z 996.86,A -85,B 0,C 180,E1 15619.043,E2 15619.043} C_VEL
LIN {X 0,Y 343.514,Z 974.48,A -85,B 0,C 180,E1 15617.754,E2 15617.754} C_VEL
LIN {X 0,Y 346.587,Z 949.754,A -85,B 0,C 180,E1 15616.653,E2 15616.653} C_VEL
LIN {X 0,Y 349.409,Z 920.575,A -85,B 0,C 180,E1 15615.72,E2 15615.72} C_VEL
LIN {X 0,Y 364.147,Z 759.422,A -85,B 0,C 180,E1 15611.252,E2 15611.252} C_VEL
LIN {X 0,Y 347.296,Z 728.853,A -85,B 0,C 180,E1 15608.009,E2 15608.009} C_VEL
LIN {X 0,Y 331.647,Z 702.081,A -85,B 0,C 180,E1 15604.687,E2 15604.687} C_VEL
LIN {X 0,Y 318.273,Z 680.493,A -85,B 0,C 180,E1 15601.594,E2 15601.594} C_VEL
LIN {X 0,Y 312.22,Z 671.136,A -85,B 0,C 180,E1 15600.108,E2 15600.108} C_VEL
LIN {X 0,Y 309.844,Z 667.191,A -85,B 0,C 180,E1 15599.483,E2 15599.483} C_VEL
LIN {X 0,Y 307.812,Z 664.087,A -85,B 0,C 180,E1 15598.95,E2 15598.95} C_VEL
LIN {X 0,Y 307.395,Z 662.372,A -85,B 0,C 180,E1 15598.78,E2 15598.78} C_VEL
LIN {X 0,Y 307.358,Z 662.388,A -85,B 0,C 180,E1 15594.201,E2 15594.201} C_VEL
LIN {X 0,Y 307.366,Z 662.38,A -85,B 0,C 180,E1 15589.579,E2 15589.579} C_VEL
LIN {X 0,Y 307.382,Z 662.375,A -85,B 0,C 180,E1 15585.086,E2 15585.086} C_VEL
LIN {X 0,Y 307.393,Z 662.379,A -85,B 0,C 180,E1 15580.687,E2 15580.687} C_VEL
LIN {X 0,Y 307.349,Z 662.385,A -85,B 0,C 180,E1 15576.165,E2 15576.165} C_VEL
LIN {X 0,Y 307.349,Z 662.366,A -85,B 0,C 180,E1 15571.494,E2 15571.494} C_VEL
LIN {X 0,Y 307.391,Z 662.359,A -85,B 0,C 180,E1 15567.206,E2 15567.206} C_VEL
LIN {X 0,Y 307.408,Z 662.375,A -85,B 0,C 180,E1 15562.715,E2 15562.715} C_VEL
LIN {X 0,Y 307.358,Z 662.351,A -85,B 0,C 180,E1 15558.176,E2 15558.176} C_VEL
LIN {X 0,Y 307.338,Z 662.381,A -85,B 0,C 180,E1 15553.561,E2 15553.561} C_VEL
LIN {X 0,Y 307.395,Z 662.374,A -85,B 0,C 180,E1 15549.038,E2 15549.038} C_VEL
LIN {X 0,Y 307.392,Z 662.376,A -85,B 0,C 180,E1 15544.576,E2 15544.576} C_VEL
LIN {X 0,Y 307.386,Z 662.379,A -85,B 0,C 180,E1 15540.156,E2 15540.156} C_VEL
LIN {X 0,Y 307.352,Z 662.453,A -85,B 0,C 180,E1 15537.66,E2 15537.66} C_VEL
LIN {X 0,Y 316.465,Z 688.448,A -85,B 0,C 180,E1 15533.668,E2 15533.668} C_VEL
LIN {X 0,Y 323.409,Z 710.876,A -85,B 0,C 180,E1 15530.443,E2 15530.443} C_VEL
LIN {X 0,Y 328.305,Z 729.104,A -85,B 0,C 180,E1 15527.992,E2 15527.992} C_VEL
LIN {X 0,Y 324.7,Z 771.296,A -85,B 0,C 180,E1 15523.607,E2 15523.607} C_VEL
LIN {X 0,Y 321.071,Z 815.839,A -85,B 0,C 180,E1 15518.976,E2 15518.976} C_VEL
LIN {X 0,Y 318.303,Z 851.655,A -85,B 0,C 180,E1 15515.246,E2 15515.246} C_VEL
LIN {X 0,Y 317.62,Z 856.411,A -85,B 0,C 180,E1 15514.82,E2 15514.82} C_VEL
LIN {X 0,Y 312.647,Z 985.538,A -85,B 0,C 180,E1 15510.656,E2 15510.656} C_VEL
LIN {X 0,Y 312.185,Z 1007.105,A -85,B 0,C 180,E1 15509.837,E2 15509.837} C_VEL
LIN {X 0,Y 311.917,Z 1014.671,A -85,B 0,C 180,E1 15509.444,E2 15509.444} C_VEL
LIN {X 0,Y 310.627,Z 1021.994,A -85,B 0,C 180,E1 15509.033,E2 15509.033} C_VEL
LIN {X 0,Y 304.416,Z 1037.795,A -85,B 0,C 180,E1 15507.951,E2 15507.951} C_VEL
LIN {X 0,Y 302.554,Z 1044.666,A -85,B 0,C 180,E1 15507.351,E2 15507.351} C_VEL
LIN {X 0,Y 302.34,Z 1046.616,A -85,B 0,C 180,E1 15507.162,E2 15507.162} C_VEL
LIN {X 0,Y 301.3,Z 1061.57,A -85,B 0,C 180,E1 15505.454,E2 15505.454} C_VEL
LIN {X 0,Y 300.265,Z 1075.604,A -85,B 0,C 180,E1 15503.444,E2 15503.444} C_VEL
LIN {X 0,Y 299.275,Z 1088.996,A -85,B 0,C 180,E1 15501.044,E2 15501.044} C_VEL
LIN {X 0,Y 298.572,Z 1100.071,A -85,B 0,C 180,E1 15498.546,E2 15498.546} C_VEL
LIN {X 0,Y 298.152,Z 1109.318,A -85,B 0,C 180,E1 15495.957,E2 15495.957} C_VEL
LIN {X 0,Y 298.03,Z 1117.531,A -85,B 0,C 180,E1 15492.986,E2 15492.986} C_VEL
LIN {X 0,Y 298.279,Z 1123.208,A -85,B 0,C 180,E1 15490.229,E2 15490.229} C_VEL
LIN {X 0,Y 299.02,Z 1127.65,A -85,B 0,C 180,E1 15487.103,E2 15487.103} C_VEL
LIN {X 0,Y 300.23,Z 1130.012,A -85,B 0,C 180,E1 15484.198,E2 15484.198} C_VEL
LIN {X 0,Y 302.11,Z 1130.646,A -85,B 0,C 180,E1 15481.134,E2 15481.134} C_VEL
LIN {X 0,Y 304.475,Z 1129.548,A -85,B 0,C 180,E1 15478.302,E2 15478.302} C_VEL
LIN {X 0,Y 307.637,Z 1126.441,A -85,B 0,C 180,E1 15475.335,E2 15475.335} C_VEL
LIN {X 0,Y 311.221,Z 1121.704,A -85,B 0,C 180,E1 15472.613,E2 15472.613} C_VEL
LIN {X 0,Y 315.364,Z 1114.966,A -85,B 0,C 180,E1 15469.954,E2 15469.954} C_VEL
LIN {X 0,Y 319.717,Z 1106.715,A -85,B 0,C 180,E1 15467.534,E2 15467.534} C_VEL
LIN {X 0,Y 324.499,Z 1096.134,A -85,B 0,C 180,E1 15465.178,E2 15465.178} C_VEL
LIN {X 0,Y 328.881,Z 1084.714,A -85,B 0,C 180,E1 15463.209,E2 15463.209} C_VEL
LIN {X 0,Y 333.11,Z 1071.879,A -85,B 0,C 180,E1 15461.444,E2 15461.444} C_VEL
LIN {X 0,Y 337.314,Z 1056.403,A -85,B 0,C 180,E1 15459.794,E2 15459.794} C_VEL
LIN {X 0,Y 340.782,Z 1040.193,A -85,B 0,C 180,E1 15458.48,E2 15458.48} C_VEL
LIN {X 0,Y 343.629,Z 1021.968,A -85,B 0,C 180,E1 15457.387,E2 15457.387} C_VEL
LIN {X 0,Y 346.853,Z 992.644,A -85,B 0,C 180,E1 15456.189,E2 15456.189} C_VEL
LIN {X 0,Y 362.049,Z 883.75,A -85,B 0,C 180,E1 15452.576,E2 15452.576} C_VEL
LIN {X 0,Y 362.307,Z 878.467,A -85,B 0,C 180,E1 15452.106,E2 15452.106} C_VEL
LIN {X 0,Y 374.807,Z 831.535,A -85,B 0,C 180,E1 15447.025,E2 15447.025} C_VEL
LIN {X 0,Y 387.599,Z 791.343,A -85,B 0,C 180,E1 15442.68,E2 15442.68} C_VEL
LIN {X 0,Y 387.769,Z 790.071,A -85,B 0,C 180,E1 15442.182,E2 15442.182} C_VEL
LIN {X 0,Y 384.61,Z 796.726,A -85,B 0,C 180,E1 15441.848,E2 15441.848} C_VEL
LIN {X 0,Y 378.493,Z 810.437,A -85,B 0,C 180,E1 15441.194,E2 15441.194} C_VEL
LIN {X 0,Y 376.097,Z 815.959,A -85,B 0,C 180,E1 15440.919,E2 15440.919} C_VEL
LIN {X 0,Y 370.539,Z 829.057,A -85,B 0,C 180,E1 15440.265,E2 15440.265} C_VEL
LIN {X 0,Y 368.269,Z 834.682,A -85,B 0,C 180,E1 15439.961,E2 15439.961} C_VEL
LIN {X 0,Y 363.221,Z 847.356,A -85,B 0,C 180,E1 15439.319,E2 15439.319} C_VEL
LIN {X 0,Y 360.663,Z 854.041,A -85,B 0,C 180,E1 15438.921,E2 15438.921} C_VEL
LIN {X 0,Y 355.905,Z 867.103,A -85,B 0,C 180,E1 15438.25,E2 15438.25} C_VEL
LIN {X 0,Y 353.512,Z 873.88,A -85,B 0,C 180,E1 15437.817,E2 15437.817} C_VEL
LIN {X 0,Y 349.058,Z 886.571,A -85,B 0,C 180,E1 15437.161,E2 15437.161} C_VEL
LIN {X 0,Y 346.943,Z 893.956,A -85,B 0,C 180,E1 15436.66,E2 15436.66} C_VEL
LIN {X 0,Y 339.402,Z 975.768,A -85,B 0,C 180,E1 15434.204,E2 15434.204} C_VEL
LIN {X 0,Y 336.11,Z 1000.417,A -85,B 0,C 180,E1 15433.17,E2 15433.17} C_VEL
LIN {X 0,Y 332.12,Z 1024.661,A -85,B 0,C 180,E1 15431.821,E2 15431.821} C_VEL
LIN {X 0,Y 327.787,Z 1047.739,A -85,B 0,C 180,E1 15430.174,E2 15430.174} C_VEL
LIN {X 0,Y 323.368,Z 1068.852,A -85,B 0,C 180,E1 15428.31,E2 15428.31} C_VEL
LIN {X 0,Y 318.802,Z 1089.24,A -85,B 0,C 180,E1 15426.128,E2 15426.128} C_VEL
LIN {X 0,Y 314.232,Z 1108.743,A -85,B 0,C 180,E1 15423.615,E2 15423.615} C_VEL
LIN {X 0,Y 309.968,Z 1126.647,A -85,B 0,C 180,E1 15420.854,E2 15420.854} C_VEL
LIN {X 0,Y 306.11,Z 1143.031,A -85,B 0,C 180,E1 15417.843,E2 15417.843} C_VEL
LIN {X 0,Y 302.801,Z 1157.859,A -85,B 0,C 180,E1 15414.583,E2 15414.583} C_VEL
LIN {X 0,Y 300.159,Z 1170.946,A -85,B 0,C 180,E1 15411.127,E2 15411.127} C_VEL
LIN {X 0,Y 298.273,Z 1182.212,A -85,B 0,C 180,E1 15407.557,E2 15407.557} C_VEL
LIN {X 0,Y 297.13,Z 1191.479,A -85,B 0,C 180,E1 15404.019,E2 15404.019} C_VEL
LIN {X 0,Y 296.588,Z 1198.873,A -85,B 0,C 180,E1 15400.486,E2 15400.486} C_VEL
LIN {X 0,Y 296.471,Z 1204.945,A -85,B 0,C 180,E1 15396.776,E2 15396.776} C_VEL
LIN {X 0,Y 296.52,Z 1208.943,A -85,B 0,C 180,E1 15393.451,E2 15393.451} C_VEL
LIN {X 0,Y 296.481,Z 1211.798,A -85,B 0,C 180,E1 15389.804,E2 15389.804} C_VEL
LIN {X 0,Y 296.27,Z 1213.038,A -85,B 0,C 180,E1 15386.515,E2 15386.515} C_VEL
LIN {X 0,Y 296.096,Z 1213.092,A -85,B 0,C 180,E1 15382.625,E2 15382.625} C_VEL
LIN {X 0,Y 296.432,Z 1211.443,A -85,B 0,C 180,E1 15378.518,E2 15378.518} C_VEL
LIN {X 0,Y 297.885,Z 1207.902,A -85,B 0,C 180,E1 15374.021,E2 15374.021} C_VEL
LIN {X 0,Y 300.786,Z 1202.629,A -85,B 0,C 180,E1 15369.569,E2 15369.569} C_VEL
LIN {X 0,Y 305.55,Z 1195.184,A -85,B 0,C 180,E1 15365.028,E2 15365.028} C_VEL
LIN {X 0,Y 312.223,Z 1185.885,A -85,B 0,C 180,E1 15360.658,E2 15360.658} C_VEL
LIN {X 0,Y 321.664,Z 1173.799,A -85,B 0,C 180,E1 15356.189,E2 15356.189} C_VEL
LIN {X 0,Y 333.281,Z 1159.846,A -85,B 0,C 180,E1 15352.1,E2 15352.1} C_VEL
LIN {X 0,Y 346.893,Z 1144.326,A -85,B 0,C 180,E1 15348.472,E2 15348.472} C_VEL
LIN {X 0,Y 361.794,Z 1127.983,A -85,B 0,C 180,E1 15345.412,E2 15345.412} C_VEL
LIN {X 0,Y 371.807,Z 1117.295,A -85,B 0,C 180,E1 15343.724,E2 15343.724} C_VEL
LIN {X 0,Y 356.548,Z 1132.084,A -85,B 0,C 180,E1 15340.803,E2 15340.803} C_VEL
LIN {X 0,Y 342.533,Z 1145.713,A -85,B 0,C 180,E1 15337.389,E2 15337.389} C_VEL
LIN {X 0,Y 330.445,Z 1157.502,A -85,B 0,C 180,E1 15333.628,E2 15333.628} C_VEL
LIN {X 0,Y 320.653,Z 1167.035,A -85,B 0,C 180,E1 15329.727,E2 15329.727} C_VEL
LIN {X 0,Y 312.64,Z 1174.829,A -85,B 0,C 180,E1 15325.583,E2 15325.583} C_VEL
LIN {X 0,Y 306.161,Z 1181.052,A -85,B 0,C 180,E1 15321.058,E2 15321.058} C_VEL
LIN {X 0,Y 301.831,Z 1185.076,A -85,B 0,C 180,E1 15316.755,E2 15316.755} C_VEL
LIN {X 0,Y 298.923,Z 1187.372,A -85,B 0,C 180,E1 15312.365,E2 15312.365} C_VEL
LIN {X 0,Y 297.278,Z 1187.928,A -85,B 0,C 180,E1 15308.125,E2 15308.125} C_VEL
LIN {X 0,Y 296.518,Z 1186.998,A -85,B 0,C 180,E1 15304.065,E2 15304.065} C_VEL
LIN {X 0,Y 296.244,Z 1184.751,A -85,B 0,C 180,E1 15300.391,E2 15300.391} C_VEL
LIN {X 0,Y 296.194,Z 1180.967,A -85,B 0,C 180,E1 15296.521,E2 15296.521} C_VEL
LIN {X 0,Y 296.344,Z 1176.179,A -85,B 0,C 180,E1 15293.028,E2 15293.028} C_VEL
LIN {X 0,Y 296.893,Z 1169.179,A -85,B 0,C 180,E1 15289.133,E2 15289.133} C_VEL
LIN {X 0,Y 297.938,Z 1160.827,A -85,B 0,C 180,E1 15285.426,E2 15285.426} C_VEL
LIN {X 0,Y 299.64,Z 1150.534,A -85,B 0,C 180,E1 15281.724,E2 15281.724} C_VEL
LIN {X 0,Y 301.967,Z 1138.798,A -85,B 0,C 180,E1 15278.236,E2 15278.236} C_VEL
LIN {X 0,Y 305.042,Z 1124.933,A -85,B 0,C 180,E1 15274.783,E2 15274.783} C_VEL
LIN {X 0,Y 308.558,Z 1110.05,A -85,B 0,C 180,E1 15271.663,E2 15271.663} C_VEL
LIN {X 0,Y 312.478,Z 1093.775,A -85,B 0,C 180,E1 15268.782,E2 15268.782} C_VEL
LIN {X 0,Y 316.846,Z 1075.318,A -85,B 0,C 180,E1 15266.049,E2 15266.049} C_VEL
LIN {X 0,Y 321.273,Z 1055.918,A -85,B 0,C 180,E1 15263.643,E2 15263.643} C_VEL
LIN {X 0,Y 325.766,Z 1034.834,A -85,B 0,C 180,E1 15261.465,E2 15261.465} C_VEL
LIN {X 0,Y 330.203,Z 1012.117,A -85,B 0,C 180,E1 15259.543,E2 15259.543} C_VEL
LIN {X 0,Y 334.119,Z 989.354,A -85,B 0,C 180,E1 15257.988,E2 15257.988} C_VEL
LIN {X 0,Y 337.542,Z 965.885,A -85,B 0,C 180,E1 15256.718,E2 15256.718} C_VEL
LIN {X 0,Y 340.417,Z 941.956,A -85,B 0,C 180,E1 15255.735,E2 15255.735} C_VEL
LIN {X 0,Y 357.384,Z 762.229,A -85,B 0,C 180,E1 15250.581,E2 15250.581} C_VEL
LIN {X 0,Y 340.885,Z 732.153,A -85,B 0,C 180,E1 15247.308,E2 15247.308} C_VEL
LIN {X 0,Y 324.619,Z 704.326,A -85,B 0,C 180,E1 15243.754,E2 15243.754} C_VEL
LIN {X 0,Y 310.831,Z 682.109,A -85,B 0,C 180,E1 15240.443,E2 15240.443} C_VEL
LIN {X 0,Y 304.67,Z 672.572,A -85,B 0,C 180,E1 15238.847,E2 15238.847} C_VEL
LIN {X 0,Y 301.922,Z 668.216,A -85,B 0,C 180,E1 15238.108,E2 15238.108} C_VEL
LIN {X 0,Y 299.881,Z 665.103,A -85,B 0,C 180,E1 15237.559,E2 15237.559} C_VEL
LIN {X 0,Y 299.463,Z 663.369,A -85,B 0,C 180,E1 15237.369,E2 15237.369} C_VEL
LIN {X 0,Y 299.395,Z 663.366,A -85,B 0,C 180,E1 15232.796,E2 15232.796} C_VEL
LIN {X 0,Y 299.424,Z 663.356,A -85,B 0,C 180,E1 15228.096,E2 15228.096} C_VEL
LIN {X 0,Y 299.463,Z 663.347,A -85,B 0,C 180,E1 15223.702,E2 15223.702} C_VEL
LIN {X 0,Y 299.456,Z 663.349,A -85,B 0,C 180,E1 15219.031,E2 15219.031} C_VEL
LIN {X 0,Y 299.403,Z 663.37,A -85,B 0,C 180,E1 15214.6,E2 15214.6} C_VEL
LIN {X 0,Y 299.419,Z 663.371,A -85,B 0,C 180,E1 15209.811,E2 15209.811} C_VEL
LIN {X 0,Y 299.453,Z 663.341,A -85,B 0,C 180,E1 15205.406,E2 15205.406} C_VEL
LIN {X 0,Y 299.443,Z 663.358,A -85,B 0,C 180,E1 15200.973,E2 15200.973} C_VEL
LIN {X 0,Y 299.421,Z 663.359,A -85,B 0,C 180,E1 15196.484,E2 15196.484} C_VEL
LIN {X 0,Y 299.422,Z 663.369,A -85,B 0,C 180,E1 15191.91,E2 15191.91} C_VEL
LIN {X 0,Y 299.464,Z 663.363,A -85,B 0,C 180,E1 15187.216,E2 15187.216} C_VEL
LIN {X 0,Y 299.444,Z 663.369,A -85,B 0,C 180,E1 15182.564,E2 15182.564} C_VEL
LIN {X 0,Y 299.412,Z 663.377,A -85,B 0,C 180,E1 15178.445,E2 15178.445} C_VEL
LIN {X 0,Y 308.541,Z 689.322,A -85,B 0,C 180,E1 15174.319,E2 15174.319} C_VEL
LIN {X 0,Y 315.417,Z 711.207,A -85,B 0,C 180,E1 15171.125,E2 15171.125} C_VEL
LIN {X 0,Y 320.779,Z 730.854,A -85,B 0,C 180,E1 15168.403,E2 15168.403} C_VEL
LIN {X 0,Y 317.133,Z 772.172,A -85,B 0,C 180,E1 15164.044,E2 15164.044} C_VEL
LIN {X 0,Y 313.378,Z 816.776,A -85,B 0,C 180,E1 15159.34,E2 15159.34} C_VEL
LIN {X 0,Y 310.59,Z 852.018,A -85,B 0,C 180,E1 15155.635,E2 15155.635} C_VEL
LIN {X 0,Y 309.82,Z 857.346,A -85,B 0,C 180,E1 15155.148,E2 15155.148} C_VEL
LIN {X 0,Y 304.731,Z 985.54,A -85,B 0,C 180,E1 15150.872,E2 15150.872} C_VEL
LIN {X 0,Y 304.251,Z 1007.476,A -85,B 0,C 180,E1 15150.025,E2 15150.025} C_VEL
LIN {X 0,Y 303.549,Z 1024.748,A -85,B 0,C 180,E1 15149.01,E2 15149.01} C_VEL
LIN {X 0,Y 302.668,Z 1041.416,A -85,B 0,C 180,E1 15147.667,E2 15147.667} C_VEL
LIN {X 0,Y 302.34,Z 1046.616,A -85,B 0,C 180,E1 15147.162,E2 15147.162} C_VEL
LIN {X 0,Y 300.911,Z 1053.345,A -85,B 0,C 180,E1 15146.48,E2 15146.48} C_VEL
LIN {X 0,Y 295.227,Z 1065.759,A -85,B 0,C 180,E1 15144.997,E2 15144.997} C_VEL
LIN {X 0,Y 292.71,Z 1072.704,A -85,B 0,C 180,E1 15144.011,E2 15144.011} C_VEL
LIN {X 0,Y 292.311,Z 1075.296,A -85,B 0,C 180,E1 15143.611,E2 15143.611} C_VEL
LIN {X 0,Y 291.321,Z 1088.537,A -85,B 0,C 180,E1 15141.224,E2 15141.224} C_VEL
LIN {X 0,Y 290.635,Z 1099.168,A -85,B 0,C 180,E1 15138.863,E2 15138.863} C_VEL
LIN {X 0,Y 290.153,Z 1109.542,A -85,B 0,C 180,E1 15135.973,E2 15135.973} C_VEL
LIN {X 0,Y 290.029,Z 1117.371,A -85,B 0,C 180,E1 15133.148,E2 15133.148} C_VEL
LIN {X 0,Y 290.304,Z 1123.763,A -85,B 0,C 180,E1 15130.112,E2 15130.112} C_VEL
LIN {X 0,Y 291.166,Z 1128.635,A -85,B 0,C 180,E1 15126.701,E2 15126.701} C_VEL
LIN {X 0,Y 292.538,Z 1131.131,A -85,B 0,C 180,E1 15123.635,E2 15123.635} C_VEL
LIN {X 0,Y 294.683,Z 1131.807,A -85,B 0,C 180,E1 15120.385,E2 15120.385} C_VEL
LIN {X 0,Y 297.273,Z 1130.674,A -85,B 0,C 180,E1 15117.49,E2 15117.49} C_VEL
LIN {X 0,Y 300.714,Z 1127.56,A -85,B 0,C 180,E1 15114.463,E2 15114.463} C_VEL
LIN {X 0,Y 304.58,Z 1122.818,A -85,B 0,C 180,E1 15111.691,E2 15111.691} C_VEL
LIN {X 0,Y 309.031,Z 1116.108,A -85,B 0,C 180,E1 15108.991,E2 15108.991} C_VEL
LIN {X 0,Y 313.676,Z 1107.861,A -85,B 0,C 180,E1 15106.54,E2 15106.54} C_VEL
LIN {X 0,Y 318.769,Z 1097.31,A -85,B 0,C 180,E1 15104.16,E2 15104.16} C_VEL
LIN {X 0,Y 323.629,Z 1085.419,A -85,B 0,C 180,E1 15102.091,E2 15102.091} C_VEL
LIN {X 0,Y 328.116,Z 1072.515,A -85,B 0,C 180,E1 15100.318,E2 15100.318} C_VEL
LIN {X 0,Y 332.362,Z 1057.819,A -85,B 0,C 180,E1 15098.742,E2 15098.742} C_VEL
LIN {X 0,Y 336.039,Z 1041.813,A -85,B 0,C 180,E1 15097.425,E2 15097.425} C_VEL
LIN {X 0,Y 339.142,Z 1023.371,A -85,B 0,C 180,E1 15096.3,E2 15096.3} C_VEL
LIN {X 0,Y 342.609,Z 994.237,A -85,B 0,C 180,E1 15095.088,E2 15095.088} C_VEL
LIN {X 0,Y 358.578,Z 885.978,A -85,B 0,C 180,E1 15091.468,E2 15091.468} C_VEL
LIN {X 0,Y 358.936,Z 879.84,A -85,B 0,C 180,E1 15090.912,E2 15090.912} C_VEL
LIN {X 0,Y 372.026,Z 834,A -85,B 0,C 180,E1 15085.915,E2 15085.915} C_VEL
LIN {X 0,Y 381.715,Z 805.031,A -85,B 0,C 180,E1 15082.751,E2 15082.751} C_VEL
LIN {X 0,Y 375.678,Z 817.877,A -85,B 0,C 180,E1 15082.102,E2 15082.102} C_VEL
LIN {X 0,Y 369.6,Z 831.711,A -85,B 0,C 180,E1 15081.425,E2 15081.425} C_VEL
LIN {X 0,Y 367.22,Z 837.241,A -85,B 0,C 180,E1 15081.141,E2 15081.141} C_VEL
LIN {X 0,Y 361.697,Z 850.482,A -85,B 0,C 180,E1 15080.464,E2 15080.464} C_VEL
LIN {X 0,Y 359.488,Z 856.078,A -85,B 0,C 180,E1 15080.141,E2 15080.141} C_VEL
LIN {X 0,Y 354.088,Z 869.909,A -85,B 0,C 180,E1 15079.426,E2 15079.426} C_VEL
LIN {X 0,Y 352.025,Z 875.434,A -85,B 0,C 180,E1 15079.069,E2 15079.069} C_VEL
LIN {X 0,Y 347.094,Z 888.986,A -85,B 0,C 180,E1 15078.374,E2 15078.374} C_VEL
LIN {X 0,Y 344.655,Z 896.645,A -85,B 0,C 180,E1 15077.879,E2 15077.879} C_VEL
LIN {X 0,Y 338.017,Z 930.403,A -85,B 0,C 180,E1 15076.566,E2 15076.566} C_VEL
LIN {X 0,Y 334.907,Z 948.716,A -85,B 0,C 180,E1 15075.697,E2 15075.697} C_VEL
LIN {X 0,Y 331.697,Z 980.42,A -85,B 0,C 180,E1 15074.641,E2 15074.641} C_VEL
LIN {X 0,Y 328.247,Z 1004.301,A -85,B 0,C 180,E1 15073.562,E2 15073.562} C_VEL
LIN {X 0,Y 324.355,Z 1027.083,A -85,B 0,C 180,E1 15072.22,E2 15072.22} C_VEL
LIN {X 0,Y 319.956,Z 1049.679,A -85,B 0,C 180,E1 15070.539,E2 15070.539} C_VEL
LIN {X 0,Y 316.473,Z 1067.558,A -85,B 0,C 180,E1 15069.069,E2 15069.069} C_VEL
LIN {X 0,Y 313.491,Z 1083.012,A -85,B 0,C 180,E1 15067.643,E2 15067.643} C_VEL
LIN {X 0,Y 310.017,Z 1098.929,A -85,B 0,C 180,E1 15065.826,E2 15065.826} C_VEL
LIN {X 0,Y 305.82,Z 1116.097,A -85,B 0,C 180,E1 15063.426,E2 15063.426} C_VEL
LIN {X 0,Y 301.768,Z 1131.439,A -85,B 0,C 180,E1 15060.789,E2 15060.789} C_VEL
LIN {X 0,Y 298.143,Z 1144.797,A -85,B 0,C 180,E1 15058,E2 15058} C_VEL
LIN {X 0,Y 292.884,Z 1166.97,A -85,B 0,C 180,E1 15052.265,E2 15052.265} C_VEL
LIN {X 0,Y 290.763,Z 1178.733,A -85,B 0,C 180,E1 15048.648,E2 15048.648} C_VEL
LIN {X 0,Y 289.408,Z 1188.43,A -85,B 0,C 180,E1 15045.015,E2 15045.015} C_VEL
LIN {X 0,Y 288.69,Z 1196.781,A -85,B 0,C 180,E1 15041.181,E2 15041.181} C_VEL
LIN {X 0,Y 288.505,Z 1202.973,A -85,B 0,C 180,E1 15037.565,E2 15037.565} C_VEL
LIN {X 0,Y 288.556,Z 1207.536,A -85,B 0,C 180,E1 15033.971,E2 15033.971} C_VEL
LIN {X 0,Y 288.555,Z 1210.353,A -85,B 0,C 180,E1 15030.791,E2 15030.791} C_VEL
LIN {X 0,Y 288.338,Z 1212.252,A -85,B 0,C 180,E1 15027.16,E2 15027.16} C_VEL
LIN {X 0,Y 288.114,Z 1212.68,A -85,B 0,C 180,E1 15023.421,E2 15023.421} C_VEL
LIN {X 0,Y 288.313,Z 1211.712,A -85,B 0,C 180,E1 15019.204,E2 15019.204} C_VEL
LIN {X 0,Y 289.52,Z 1208.927,A -85,B 0,C 180,E1 15014.781,E2 15014.781} C_VEL
LIN {X 0,Y 292.358,Z 1204.098,A -85,B 0,C 180,E1 15009.998,E2 15009.998} C_VEL
LIN {X 0,Y 297.027,Z 1197.458,A -85,B 0,C 180,E1 15005.326,E2 15005.326} C_VEL
LIN {X 0,Y 303.976,Z 1188.607,A -85,B 0,C 180,E1 15000.649,E2 15000.649} C_VEL
LIN {X 0,Y 313.088,Z 1177.823,A -85,B 0,C 180,E1 14996.239,E2 14996.239} C_VEL
LIN {X 0,Y 324.877,Z 1164.751,A -85,B 0,C 180,E1 14992.006,E2 14992.006} C_VEL
LIN {X 0,Y 338.989,Z 1149.891,A -85,B 0,C 180,E1 14988.191,E2 14988.191} C_VEL
LIN {X 0,Y 354.695,Z 1134.04,A -85,B 0,C 180,E1 14984.96,E2 14984.96} C_VEL
LIN {X 0,Y 362.229,Z 1126.606,A -85,B 0,C 180,E1 14983.641,E2 14983.641} C_VEL
LIN {X 0,Y 346.438,Z 1140.623,A -85,B 0,C 180,E1 14980.5,E2 14980.5} C_VEL
LIN {X 0,Y 332.051,Z 1153.38,A -85,B 0,C 180,E1 14976.819,E2 14976.819} C_VEL
LIN {X 0,Y 319.546,Z 1164.458,A -85,B 0,C 180,E1 14972.674,E2 14972.674} C_VEL
LIN {X 0,Y 309.243,Z 1173.524,A -85,B 0,C 180,E1 14968.173,E2 14968.173} C_VEL
LIN {X 0,Y 301.55,Z 1180.131,A -85,B 0,C 180,E1 14963.658,E2 14963.658} C_VEL
LIN {X 0,Y 295.988,Z 1184.696,A -85,B 0,C 180,E1 14959.132,E2 14959.132} C_VEL
LIN {X 0,Y 292.133,Z 1187.511,A -85,B 0,C 180,E1 14954.473,E2 14954.473} C_VEL
LIN {X 0,Y 289.942,Z 1188.547,A -85,B 0,C 180,E1 14950.134,E2 14950.134} C_VEL
LIN {X 0,Y 288.803,Z 1187.945,A -85,B 0,C 180,E1 14945.966,E2 14945.966} C_VEL
LIN {X 0,Y 288.321,Z 1185.879,A -85,B 0,C 180,E1 14941.793,E2 14941.793} C_VEL
LIN {X 0,Y 288.19,Z 1182.837,A -85,B 0,C 180,E1 14938.215,E2 14938.215} C_VEL
LIN {X 0,Y 288.268,Z 1177.948,A -85,B 0,C 180,E1 14934.231,E2 14934.231} C_VEL
LIN {X 0,Y 288.651,Z 1171.801,A -85,B 0,C 180,E1 14930.433,E2 14930.433} C_VEL
LIN {X 0,Y 289.513,Z 1163.853,A -85,B 0,C 180,E1 14926.625,E2 14926.625} C_VEL
LIN {X 0,Y 291.121,Z 1153.553,A -85,B 0,C 180,E1 14922.619,E2 14922.619} C_VEL
LIN {X 0,Y 293.3,Z 1142.387,A -85,B 0,C 180,E1 14919.03,E2 14919.03} C_VEL
LIN {X 0,Y 296.234,Z 1129.127,A -85,B 0,C 180,E1 14915.475,E2 14915.475} C_VEL
LIN {X 0,Y 299.806,Z 1114.02,A -85,B 0,C 180,E1 14912.109,E2 14912.109} C_VEL
LIN {X 0,Y 303.717,Z 1098.006,A -85,B 0,C 180,E1 14909.103,E2 14909.103} C_VEL
LIN {X 0,Y 308.242,Z 1079.498,A -85,B 0,C 180,E1 14906.183,E2 14906.183} C_VEL
LIN {X 0,Y 312.785,Z 1060.263,A -85,B 0,C 180,E1 14903.647,E2 14903.647} C_VEL
LIN {X 0,Y 317.334,Z 1039.896,A -85,B 0,C 180,E1 14901.406,E2 14901.406} C_VEL
LIN {X 0,Y 321.866,Z 1017.806,A -85,B 0,C 180,E1 14899.403,E2 14899.403} C_VEL
LIN {X 0,Y 326.169,Z 994.146,A -85,B 0,C 180,E1 14897.674,E2 14897.674} C_VEL
LIN {X 0,Y 329.875,Z 970.056,A -85,B 0,C 180,E1 14896.29,E2 14896.29} C_VEL
LIN {X 0,Y 332.964,Z 945.501,A -85,B 0,C 180,E1 14895.219,E2 14895.219} C_VEL
LIN {X 0,Y 338.185,Z 891.036,A -85,B 0,C 180,E1 14893.534,E2 14893.534} C_VEL
LIN {X 0,Y 350.601,Z 764.958,A -85,B 0,C 180,E1 14889.893,E2 14889.893} C_VEL
LIN {X 0,Y 334.878,Z 736.294,A -85,B 0,C 180,E1 14886.696,E2 14886.696} C_VEL
LIN {X 0,Y 319.355,Z 709.518,A -85,B 0,C 180,E1 14883.2,E2 14883.2} C_VEL
LIN {X 0,Y 305.871,Z 687.635,A -85,B 0,C 180,E1 14879.878,E2 14879.878} C_VEL
LIN {X 0,Y 297,Z 673.912,A -85,B 0,C 180,E1 14877.523,E2 14877.523} C_VEL
LIN {X 0,Y 293.997,Z 669.231,A -85,B 0,C 180,E1 14876.678,E2 14876.678} C_VEL
LIN {X 0,Y 291.934,Z 666.134,A -85,B 0,C 180,E1 14876.087,E2 14876.087} C_VEL
LIN {X 0,Y 291.504,Z 664.349,A -85,B 0,C 180,E1 14875.87,E2 14875.87} C_VEL
LIN {X 0,Y 291.472,Z 664.355,A -85,B 0,C 180,E1 14871.326,E2 14871.326} C_VEL
LIN {X 0,Y 291.491,Z 664.356,A -85,B 0,C 180,E1 14866.544,E2 14866.544} C_VEL
LIN {X 0,Y 291.514,Z 664.348,A -85,B 0,C 180,E1 14862.08,E2 14862.08} C_VEL
LIN {X 0,Y 291.493,Z 664.343,A -85,B 0,C 180,E1 14857.492,E2 14857.492} C_VEL
LIN {X 0,Y 291.467,Z 664.338,A -85,B 0,C 180,E1 14852.952,E2 14852.952} C_VEL
LIN {X 0,Y 291.491,Z 664.356,A -85,B 0,C 180,E1 14848.43,E2 14848.43} C_VEL
LIN {X 0,Y 291.516,Z 664.348,A -85,B 0,C 180,E1 14843.701,E2 14843.701} C_VEL
LIN {X 0,Y 291.483,Z 664.327,A -85,B 0,C 180,E1 14839.128,E2 14839.128} C_VEL
LIN {X 0,Y 291.484,Z 664.359,A -85,B 0,C 180,E1 14834.484,E2 14834.484} C_VEL
LIN {X 0,Y 291.5,Z 664.353,A -85,B 0,C 180,E1 14829.943,E2 14829.943} C_VEL
LIN {X 0,Y 291.516,Z 664.357,A -85,B 0,C 180,E1 14825.346,E2 14825.346} C_VEL
LIN {X 0,Y 291.486,Z 664.361,A -85,B 0,C 180,E1 14820.599,E2 14820.599} C_VEL
LIN {X 0,Y 291.49,Z 664.573,A -85,B 0,C 180,E1 14819.186,E2 14819.186} C_VEL
LIN {X 0,Y 299.696,Z 687.484,A -85,B 0,C 180,E1 14815.45,E2 14815.45} C_VEL
LIN {X 0,Y 306.82,Z 709.577,A -85,B 0,C 180,E1 14812.103,E2 14812.103} C_VEL
LIN {X 0,Y 313.006,Z 731.771,A -85,B 0,C 180,E1 14808.961,E2 14808.961} C_VEL
LIN {X 0,Y 313.138,Z 734.676,A -85,B 0,C 180,E1 14808.616,E2 14808.616} C_VEL
LIN {X 0,Y 309.226,Z 777.509,A -85,B 0,C 180,E1 14804.037,E2 14804.037} C_VEL
LIN {X 0,Y 305.41,Z 821.236,A -85,B 0,C 180,E1 14799.347,E2 14799.347} C_VEL
LIN {X 0,Y 302.702,Z 853.326,A -85,B 0,C 180,E1 14795.93,E2 14795.93} C_VEL
LIN {X 0,Y 302.008,Z 858.239,A -85,B 0,C 180,E1 14795.478,E2 14795.478} C_VEL
LIN {X 0,Y 296.817,Z 985.708,A -85,B 0,C 180,E1 14791.093,E2 14791.093} C_VEL
LIN {X 0,Y 296.305,Z 1008.035,A -85,B 0,C 180,E1 14790.203,E2 14790.203} C_VEL
LIN {X 0,Y 295.61,Z 1024.805,A -85,B 0,C 180,E1 14789.198,E2 14789.198} C_VEL
LIN {X 0,Y 294.695,Z 1041.718,A -85,B 0,C 180,E1 14787.804,E2 14787.804} C_VEL
LIN {X 0,Y 293.602,Z 1057.861,A -85,B 0,C 180,E1 14786.055,E2 14786.055} C_VEL
LIN {X 0,Y 292.576,Z 1071.767,A -85,B 0,C 180,E1 14784.158,E2 14784.158} C_VEL
LIN {X 0,Y 292.311,Z 1075.296,A -85,B 0,C 180,E1 14783.611,E2 14783.611} C_VEL
LIN {X 0,Y 290.878,Z 1081.174,A -85,B 0,C 180,E1 14782.655,E2 14782.655} C_VEL
LIN {X 0,Y 285.701,Z 1091.031,A -85,B 0,C 180,E1 14780.788,E2 14780.788} C_VEL
LIN {X 0,Y 282.941,Z 1097.495,A -85,B 0,C 180,E1 14779.337,E2 14779.337} C_VEL
LIN {X 0,Y 282.618,Z 1099.617,A -85,B 0,C 180,E1 14778.82,E2 14778.82} C_VEL
LIN {X 0,Y 282.16,Z 1109.438,A -85,B 0,C 180,E1 14776.041,E2 14776.041} C_VEL
LIN {X 0,Y 282.032,Z 1117.661,A -85,B 0,C 180,E1 14773.11,E2 14773.11} C_VEL
LIN {X 0,Y 282.327,Z 1124.25,A -85,B 0,C 180,E1 14769.989,E2 14769.989} C_VEL
LIN {X 0,Y 283.248,Z 1129.372,A -85,B 0,C 180,E1 14766.482,E2 14766.482} C_VEL
LIN {X 0,Y 284.773,Z 1132.165,A -85,B 0,C 180,E1 14763.216,E2 14763.216} C_VEL
LIN {X 0,Y 286.985,Z 1132.983,A -85,B 0,C 180,E1 14759.996,E2 14759.996} C_VEL
LIN {X 0,Y 289.94,Z 1131.967,A -85,B 0,C 180,E1 14756.833,E2 14756.833} C_VEL
LIN {X 0,Y 293.624,Z 1128.969,A -85,B 0,C 180,E1 14753.74,E2 14753.74} C_VEL
LIN {X 0,Y 297.755,Z 1124.391,A -85,B 0,C 180,E1 14750.915,E2 14750.915} C_VEL
LIN {X 0,Y 302.479,Z 1117.822,A -85,B 0,C 180,E1 14748.169,E2 14748.169} C_VEL
LIN {X 0,Y 307.404,Z 1109.772,A -85,B 0,C 180,E1 14745.684,E2 14745.684} C_VEL
LIN {X 0,Y 312.778,Z 1099.423,A -85,B 0,C 180,E1 14743.275,E2 14743.275} C_VEL
LIN {X 0,Y 317.709,Z 1088.377,A -85,B 0,C 180,E1 14741.272,E2 14741.272} C_VEL
LIN {X 0,Y 322.66,Z 1075.315,A -85,B 0,C 180,E1 14739.404,E2 14739.404} C_VEL
LIN {X 0,Y 327.298,Z 1060.455,A -85,B 0,C 180,E1 14737.759,E2 14737.759} C_VEL
LIN {X 0,Y 330.77,Z 1046.655,A -85,B 0,C 180,E1 14736.574,E2 14736.574} C_VEL
LIN {X 0,Y 333.998,Z 1030.579,A -85,B 0,C 180,E1 14735.489,E2 14735.489} C_VEL
LIN {X 0,Y 336.622,Z 1011.434,A -85,B 0,C 180,E1 14734.561,E2 14734.561} C_VEL
LIN {X 0,Y 342.627,Z 968.821,A -85,B 0,C 180,E1 14732.986,E2 14732.986} C_VEL
LIN {X 0,Y 355.395,Z 888.22,A -85,B 0,C 180,E1 14730.327,E2 14730.327} C_VEL
LIN {X 0,Y 355.873,Z 881.541,A -85,B 0,C 180,E1 14729.709,E2 14729.709} C_VEL
LIN {X 0,Y 369.975,Z 835.483,A -85,B 0,C 180,E1 14724.662,E2 14724.662} C_VEL
LIN {X 0,Y 374.605,Z 822.138,A -85,B 0,C 180,E1 14723.197,E2 14723.197} C_VEL
LIN {X 0,Y 368.087,Z 836.119,A -85,B 0,C 180,E1 14722.481,E2 14722.481} C_VEL
LIN {X 0,Y 361.495,Z 851.228,A -85,B 0,C 180,E1 14721.766,E2 14721.766} C_VEL
LIN {X 0,Y 358.43,Z 858.423,A -85,B 0,C 180,E1 14721.356,E2 14721.356} C_VEL
LIN {X 0,Y 352.895,Z 871.956,A -85,B 0,C 180,E1 14720.666,E2 14720.666} C_VEL
LIN {X 0,Y 350.342,Z 878.538,A -85,B 0,C 180,E1 14720.274,E2 14720.274} C_VEL
LIN {X 0,Y 344.998,Z 892.589,A -85,B 0,C 180,E1 14719.529,E2 14719.529} C_VEL
LIN {X 0,Y 343.392,Z 899.043,A -85,B 0,C 180,E1 14719.146,E2 14719.146} C_VEL
LIN {X 0,Y 336.419,Z 933.073,A -85,B 0,C 180,E1 14717.828,E2 14717.828} C_VEL
LIN {X 0,Y 332.755,Z 951.849,A -85,B 0,C 180,E1 14716.953,E2 14716.953} C_VEL
LIN {X 0,Y 326.942,Z 981.772,A -85,B 0,C 180,E1 14715.739,E2 14715.739} C_VEL
LIN {X 0,Y 320.774,Z 1017.778,A -85,B 0,C 180,E1 14713.893,E2 14713.893} C_VEL
LIN {X 0,Y 316.626,Z 1047.166,A -85,B 0,C 180,E1 14712.064,E2 14712.064} C_VEL
LIN {X 0,Y 313.422,Z 1065.866,A -85,B 0,C 180,E1 14710.595,E2 14710.595} C_VEL
LIN {X 0,Y 310.147,Z 1080.548,A -85,B 0,C 180,E1 14709.272,E2 14709.272} C_VEL
LIN {X 0,Y 306.179,Z 1096.418,A -85,B 0,C 180,E1 14707.505,E2 14707.505} C_VEL
LIN {X 0,Y 301.39,Z 1113.442,A -85,B 0,C 180,E1 14705.138,E2 14705.138} C_VEL
LIN {X 0,Y 296.874,Z 1128.303,A -85,B 0,C 180,E1 14702.604,E2 14702.604} C_VEL
LIN {X 0,Y 292.518,Z 1142.244,A -85,B 0,C 180,E1 14699.708,E2 14699.708} C_VEL
LIN {X 0,Y 288.667,Z 1154.565,A -85,B 0,C 180,E1 14696.537,E2 14696.537} C_VEL
LIN {X 0,Y 285.583,Z 1164.788,A -85,B 0,C 180,E1 14693.302,E2 14693.302} C_VEL
LIN {X 0,Y 284.034,Z 1171.056,A -85,B 0,C 180,E1 14691.04,E2 14691.04} C_VEL
LIN {X 0,Y 282.182,Z 1182.016,A -85,B 0,C 180,E1 14687.313,E2 14687.313} C_VEL
LIN {X 0,Y 281.049,Z 1191.548,A -85,B 0,C 180,E1 14683.368,E2 14683.368} C_VEL
LIN {X 0,Y 280.603,Z 1198.78,A -85,B 0,C 180,E1 14679.638,E2 14679.638} C_VEL
LIN {X 0,Y 280.57,Z 1204.319,A -85,B 0,C 180,E1 14675.929,E2 14675.929} C_VEL
LIN {X 0,Y 280.614,Z 1208.161,A -85,B 0,C 180,E1 14672.448,E2 14672.448} C_VEL
LIN {X 0,Y 280.497,Z 1210.78,A -85,B 0,C 180,E1 14668.772,E2 14668.772} C_VEL
LIN {X 0,Y 280.23,Z 1211.965,A -85,B 0,C 180,E1 14665.29,E2 14665.29} C_VEL
LIN {X 0,Y 280.147,Z 1212.021,A -85,B 0,C 180,E1 14661.169,E2 14661.169} C_VEL
LIN {X 0,Y 280.857,Z 1210.283,A -85,B 0,C 180,E1 14656.617,E2 14656.617} C_VEL
LIN {X 0,Y 283.099,Z 1206.612,A -85,B 0,C 180,E1 14651.676,E2 14651.676} C_VEL
LIN {X 0,Y 287.192,Z 1201.128,A -85,B 0,C 180,E1 14646.809,E2 14646.809} C_VEL
LIN {X 0,Y 293.649,Z 1193.39,A -85,B 0,C 180,E1 14641.88,E2 14641.88} C_VEL
LIN {X 0,Y 302.093,Z 1184.066,A -85,B 0,C 180,E1 14637.347,E2 14637.347} C_VEL
LIN {X 0,Y 313.853,Z 1171.941,A -85,B 0,C 180,E1 14632.746,E2 14632.746} C_VEL
LIN {X 0,Y 327.578,Z 1158.514,A -85,B 0,C 180,E1 14628.75,E2 14628.75} C_VEL
LIN {X 0,Y 343.587,Z 1143.525,A -85,B 0,C 180,E1 14625.228,E2 14625.228} C_VEL
LIN {X 0,Y 352.679,Z 1135.163,A -85,B 0,C 180,E1 14623.579,E2 14623.579} C_VEL
LIN {X 0,Y 336.276,Z 1148.447,A -85,B 0,C 180,E1 14620.187,E2 14620.187} C_VEL
LIN {X 0,Y 321.521,Z 1160.324,A -85,B 0,C 180,E1 14616.223,E2 14616.223} C_VEL
LIN {X 0,Y 309.48,Z 1169.942,A -85,B 0,C 180,E1 14612,E2 14612} C_VEL
LIN {X 0,Y 299.505,Z 1177.754,A -85,B 0,C 180,E1 14607.369,E2 14607.369} C_VEL
LIN {X 0,Y 292.179,Z 1183.254,A -85,B 0,C 180,E1 14602.754,E2 14602.754} C_VEL
LIN {X 0,Y 286.925,Z 1186.892,A -85,B 0,C 180,E1 14598.072,E2 14598.072} C_VEL
LIN {X 0,Y 283.514,Z 1188.781,A -85,B 0,C 180,E1 14593.464,E2 14593.464} C_VEL
LIN {X 0,Y 281.541,Z 1189,A -85,B 0,C 180,E1 14588.994,E2 14588.994} C_VEL
LIN {X 0,Y 280.597,Z 1187.685,A -85,B 0,C 180,E1 14584.706,E2 14584.706} C_VEL
LIN {X 0,Y 280.254,Z 1185.101,A -85,B 0,C 180,E1 14580.618,E2 14580.618} C_VEL
LIN {X 0,Y 280.191,Z 1181.142,A -85,B 0,C 180,E1 14576.731,E2 14576.731} C_VEL
LIN {X 0,Y 280.379,Z 1175.492,A -85,B 0,C 180,E1 14572.628,E2 14572.628} C_VEL
LIN {X 0,Y 280.97,Z 1168.451,A -85,B 0,C 180,E1 14568.717,E2 14568.717} C_VEL
LIN {X 0,Y 282.127,Z 1159.629,A -85,B 0,C 180,E1 14564.8,E2 14564.8} C_VEL
LIN {X 0,Y 284.021,Z 1148.922,A -85,B 0,C 180,E1 14560.894,E2 14560.894} C_VEL
LIN {X 0,Y 286.586,Z 1136.799,A -85,B 0,C 180,E1 14557.22,E2 14557.22} C_VEL
LIN {X 0,Y 289.748,Z 1123.194,A -85,B 0,C 180,E1 14553.792,E2 14553.792} C_VEL
LIN {X 0,Y 293.541,Z 1107.808,A -85,B 0,C 180,E1 14550.52,E2 14550.52} C_VEL
LIN {X 0,Y 298.059,Z 1089.822,A -85,B 0,C 180,E1 14547.315,E2 14547.315} C_VEL
LIN {X 0,Y 302.629,Z 1071.349,A -85,B 0,C 180,E1 14544.566,E2 14544.566} C_VEL
LIN {X 0,Y 307.206,Z 1052.058,A -85,B 0,C 180,E1 14542.161,E2 14542.161} C_VEL
LIN {X 0,Y 312.016,Z 1030.195,A -85,B 0,C 180,E1 14539.906,E2 14539.906} C_VEL
LIN {X 0,Y 316.607,Z 1007.141,A -85,B 0,C 180,E1 14537.976,E2 14537.976} C_VEL
LIN {X 0,Y 320.671,Z 983.685,A -85,B 0,C 180,E1 14536.407,E2 14536.407} C_VEL
LIN {X 0,Y 324.14,Z 959.968,A -85,B 0,C 180,E1 14535.166,E2 14535.166} C_VEL
LIN {X 0,Y 326.942,Z 936.098,A -85,B 0,C 180,E1 14534.229,E2 14534.229} C_VEL
LIN {X 0,Y 343.896,Z 767.85,A -85,B 0,C 180,E1 14529.202,E2 14529.202} C_VEL
LIN {X 0,Y 328.995,Z 740.552,A -85,B 0,C 180,E1 14526.078,E2 14526.078} C_VEL
LIN {X 0,Y 314.041,Z 714.658,A -85,B 0,C 180,E1 14522.637,E2 14522.637} C_VEL
LIN {X 0,Y 301.013,Z 693.324,A -85,B 0,C 180,E1 14519.34,E2 14519.34} C_VEL
LIN {X 0,Y 291.974,Z 679.324,A -85,B 0,C 180,E1 14516.877,E2 14516.877} C_VEL
LIN {X 0,Y 288.979,Z 674.768,A -85,B 0,C 180,E1 14516.015,E2 14516.015} C_VEL
LIN {X 0,Y 286.16,Z 670.314,A -85,B 0,C 180,E1 14515.174,E2 14515.174} C_VEL
LIN {X 0,Y 284.026,Z 667.274,A -85,B 0,C 180,E1 14514.548,E2 14514.548} C_VEL
LIN {X 0,Y 283.541,Z 665.356,A -85,B 0,C 180,E1 14514.315,E2 14514.315} C_VEL
LIN {X 0,Y 283.548,Z 665.346,A -85,B 0,C 180,E1 14509.575,E2 14509.575} C_VEL
LIN {X 0,Y 283.562,Z 665.337,A -85,B 0,C 180,E1 14504.919,E2 14504.919} C_VEL
LIN {X 0,Y 283.569,Z 665.343,A -85,B 0,C 180,E1 14500.363,E2 14500.363} C_VEL
LIN {X 0,Y 283.534,Z 665.352,A -85,B 0,C 180,E1 14495.669,E2 14495.669} C_VEL
LIN {X 0,Y 283.548,Z 665.338,A -85,B 0,C 180,E1 14490.811,E2 14490.811} C_VEL
LIN {X 0,Y 283.564,Z 665.317,A -85,B 0,C 180,E1 14486.161,E2 14486.161} C_VEL
LIN {X 0,Y 283.565,Z 665.342,A -85,B 0,C 180,E1 14481.69,E2 14481.69} C_VEL
LIN {X 0,Y 283.533,Z 665.332,A -85,B 0,C 180,E1 14476.959,E2 14476.959} C_VEL
LIN {X 0,Y 283.551,Z 665.344,A -85,B 0,C 180,E1 14472.177,E2 14472.177} C_VEL
LIN {X 0,Y 283.582,Z 665.343,A -85,B 0,C 180,E1 14467.401,E2 14467.401} C_VEL
LIN {X 0,Y 283.563,Z 665.347,A -85,B 0,C 180,E1 14462.685,E2 14462.685} C_VEL
LIN {X 0,Y 283.571,Z 665.407,A -85,B 0,C 180,E1 14460.021,E2 14460.021} C_VEL
LIN {X 0,Y 292.851,Z 691.405,A -85,B 0,C 180,E1 14455.715,E2 14455.715} C_VEL
LIN {X 0,Y 299.897,Z 713.568,A -85,B 0,C 180,E1 14452.284,E2 14452.284} C_VEL
LIN {X 0,Y 305.804,Z 734.958,A -85,B 0,C 180,E1 14449.227,E2 14449.227} C_VEL
LIN {X 0,Y 301.69,Z 778.459,A -85,B 0,C 180,E1 14444.509,E2 14444.509} C_VEL
LIN {X 0,Y 297.794,Z 821.683,A -85,B 0,C 180,E1 14439.806,E2 14439.806} C_VEL
LIN {X 0,Y 295.038,Z 853.314,A -85,B 0,C 180,E1 14436.37,E2 14436.37} C_VEL
LIN {X 0,Y 294.208,Z 859.033,A -85,B 0,C 180,E1 14435.825,E2 14435.825} C_VEL
LIN {X 0,Y 288.887,Z 985.695,A -85,B 0,C 180,E1 14431.3,E2 14431.3} C_VEL
LIN {X 0,Y 288.327,Z 1009.06,A -85,B 0,C 180,E1 14430.339,E2 14430.339} C_VEL
LIN {X 0,Y 287.602,Z 1026.045,A -85,B 0,C 180,E1 14429.286,E2 14429.286} C_VEL
LIN {X 0,Y 286.667,Z 1042.847,A -85,B 0,C 180,E1 14427.859,E2 14427.859} C_VEL
LIN {X 0,Y 285.554,Z 1058.958,A -85,B 0,C 180,E1 14426.063,E2 14426.063} C_VEL
LIN {X 0,Y 284.489,Z 1073.215,A -85,B 0,C 180,E1 14424.055,E2 14424.055} C_VEL
LIN {X 0,Y 283.486,Z 1086.511,A -85,B 0,C 180,E1 14421.732,E2 14421.732} C_VEL
LIN {X 0,Y 282.706,Z 1098.062,A -85,B 0,C 180,E1 14419.199,E2 14419.199} C_VEL
LIN {X 0,Y 282.618,Z 1099.617,A -85,B 0,C 180,E1 14418.82,E2 14418.82} C_VEL
LIN {X 0,Y 281.381,Z 1104.356,A -85,B 0,C 180,E1 14417.597,E2 14417.597} C_VEL
LIN {X 0,Y 276.998,Z 1111.467,A -85,B 0,C 180,E1 14415.436,E2 14415.436} C_VEL
LIN {X 0,Y 274.376,Z 1116.32,A -85,B 0,C 180,E1 14413.68,E2 14413.68} C_VEL
LIN {X 0,Y 274.04,Z 1118.415,A -85,B 0,C 180,E1 14412.86,E2 14412.86} C_VEL
LIN {X 0,Y 274.349,Z 1124.697,A -85,B 0,C 180,E1 14409.858,E2 14409.858} C_VEL
LIN {X 0,Y 275.331,Z 1130.084,A -85,B 0,C 180,E1 14406.25,E2 14406.25} C_VEL
LIN {X 0,Y 276.948,Z 1133.076,A -85,B 0,C 180,E1 14402.893,E2 14402.893} C_VEL
LIN {X 0,Y 279.135,Z 1134.169,A -85,B 0,C 180,E1 14399.79,E2 14399.79} C_VEL
LIN {X 0,Y 282.206,Z 1133.456,A -85,B 0,C 180,E1 14396.542,E2 14396.542} C_VEL
LIN {X 0,Y 285.803,Z 1131.127,A -85,B 0,C 180,E1 14393.568,E2 14393.568} C_VEL
LIN {X 0,Y 290.366,Z 1126.663,A -85,B 0,C 180,E1 14390.482,E2 14390.482} C_VEL
LIN {X 0,Y 295.313,Z 1120.585,A -85,B 0,C 180,E1 14387.68,E2 14387.68} C_VEL
LIN {X 0,Y 300.444,Z 1112.968,A -85,B 0,C 180,E1 14385.148,E2 14385.148} C_VEL
LIN {X 0,Y 305.66,Z 1104.048,A -85,B 0,C 180,E1 14382.874,E2 14382.874} C_VEL
LIN {X 0,Y 311.217,Z 1092.838,A -85,B 0,C 180,E1 14380.671,E2 14380.671} C_VEL
LIN {X 0,Y 316.158,Z 1081.191,A -85,B 0,C 180,E1 14378.863,E2 14378.863} C_VEL
LIN {X 0,Y 321.326,Z 1066.762,A -85,B 0,C 180,E1 14377.106,E2 14377.106} C_VEL
LIN {X 0,Y 325.406,Z 1052.61,A -85,B 0,C 180,E1 14375.778,E2 14375.778} C_VEL
LIN {X 0,Y 328.535,Z 1039.188,A -85,B 0,C 180,E1 14374.777,E2 14374.777} C_VEL
LIN {X 0,Y 331.32,Z 1023.807,A -85,B 0,C 180,E1 14373.878,E2 14373.878} C_VEL
LIN {X 0,Y 336.104,Z 989.741,A -85,B 0,C 180,E1 14372.477,E2 14372.477} C_VEL
LIN {X 0,Y 352.45,Z 890.477,A -85,B 0,C 180,E1 14369.159,E2 14369.159} C_VEL
LIN {X 0,Y 353.261,Z 882.749,A -85,B 0,C 180,E1 14368.42,E2 14368.42} C_VEL
LIN {X 0,Y 367.472,Z 839.265,A -85,B 0,C 180,E1 14363.629,E2 14363.629} C_VEL
LIN {X 0,Y 360.756,Z 853.897,A -85,B 0,C 180,E1 14362.957,E2 14362.957} C_VEL
LIN {X 0,Y 357.578,Z 861.009,A -85,B 0,C 180,E1 14362.57,E2 14362.57} C_VEL
LIN {X 0,Y 351.566,Z 875.178,A -85,B 0,C 180,E1 14361.845,E2 14361.845} C_VEL
LIN {X 0,Y 348.847,Z 881.721,A -85,B 0,C 180,E1 14361.484,E2 14361.484} C_VEL
LIN {X 0,Y 344.183,Z 894.047,A -85,B 0,C 180,E1 14360.844,E2 14360.844} C_VEL
LIN {X 0,Y 342.587,Z 901.329,A -85,B 0,C 180,E1 14360.429,E2 14360.429} C_VEL
LIN {X 0,Y 335.173,Z 935.573,A -85,B 0,C 180,E1 14359.113,E2 14359.113} C_VEL
LIN {X 0,Y 331.428,Z 953.567,A -85,B 0,C 180,E1 14358.283,E2 14358.283} C_VEL
LIN {X 0,Y 325.247,Z 983.697,A -85,B 0,C 180,E1 14357.071,E2 14357.071} C_VEL
LIN {X 0,Y 318.577,Z 1019.788,A -85,B 0,C 180,E1 14355.224,E2 14355.224} C_VEL
LIN {X 0,Y 313.923,Z 1048.752,A -85,B 0,C 180,E1 14353.41,E2 14353.41} C_VEL
LIN {X 0,Y 309.526,Z 1069.795,A -85,B 0,C 180,E1 14351.713,E2 14351.713} C_VEL
LIN {X 0,Y 305.04,Z 1086.465,A -85,B 0,C 180,E1 14350.095,E2 14350.095} C_VEL
LIN {X 0,Y 300.02,Z 1102.968,A -85,B 0,C 180,E1 14348.061,E2 14348.061} C_VEL
LIN {X 0,Y 294.465,Z 1119.674,A -85,B 0,C 180,E1 14345.492,E2 14345.492} C_VEL
LIN {X 0,Y 289.18,Z 1134.587,A -85,B 0,C 180,E1 14342.639,E2 14342.639} C_VEL
LIN {X 0,Y 284.319,Z 1147.843,A -85,B 0,C 180,E1 14339.491,E2 14339.491} C_VEL
LIN {X 0,Y 280.436,Z 1158.901,A -85,B 0,C 180,E1 14336.236,E2 14336.236} C_VEL
LIN {X 0,Y 277.134,Z 1168.46,A -85,B 0,C 180,E1 14332.706,E2 14332.706} C_VEL
LIN {X 0,Y 275.067,Z 1176.047,A -85,B 0,C 180,E1 14329.313,E2 14329.313} C_VEL
LIN {X 0,Y 273.495,Z 1186.811,A -85,B 0,C 180,E1 14325.153,E2 14325.153} C_VEL
LIN {X 0,Y 272.77,Z 1195.131,A -85,B 0,C 180,E1 14321.2,E2 14321.2} C_VEL
LIN {X 0,Y 272.603,Z 1201.402,A -85,B 0,C 180,E1 14317.373,E2 14317.373} C_VEL
LIN {X 0,Y 272.66,Z 1206.148,A -85,B 0,C 180,E1 14313.571,E2 14313.571} C_VEL
LIN {X 0,Y 272.626,Z 1209.166,A -85,B 0,C 180,E1 14309.997,E2 14309.997} C_VEL
LIN {X 0,Y 272.332,Z 1211.068,A -85,B 0,C 180,E1 14306.208,E2 14306.208} C_VEL
LIN {X 0,Y 272.133,Z 1211.577,A -85,B 0,C 180,E1 14301.971,E2 14301.971} C_VEL
LIN {X 0,Y 272.623,Z 1210.654,A -85,B 0,C 180,E1 14297.5,E2 14297.5} C_VEL
LIN {X 0,Y 274.49,Z 1207.828,A -85,B 0,C 180,E1 14292.618,E2 14292.618} C_VEL
LIN {X 0,Y 278.54,Z 1202.839,A -85,B 0,C 180,E1 14287.313,E2 14287.313} C_VEL
LIN {X 0,Y 284.626,Z 1196.239,A -85,B 0,C 180,E1 14282.37,E2 14282.37} C_VEL
LIN {X 0,Y 293.462,Z 1187.314,A -85,B 0,C 180,E1 14277.427,E2 14277.427} C_VEL
LIN {X 0,Y 304.765,Z 1176.578,A -85,B 0,C 180,E1 14272.864,E2 14272.864} C_VEL
LIN {X 0,Y 319.014,Z 1163.729,A -85,B 0,C 180,E1 14268.596,E2 14268.596} C_VEL
LIN {X 0,Y 335.079,Z 1149.847,A -85,B 0,C 180,E1 14264.989,E2 14264.989} C_VEL
LIN {X 0,Y 342.997,Z 1143.146,A -85,B 0,C 180,E1 14263.507,E2 14263.507} C_VEL
LIN {X 0,Y 326.056,Z 1155.615,A -85,B 0,C 180,E1 14259.865,E2 14259.865} C_VEL
LIN {X 0,Y 311.46,Z 1166.239,A -85,B 0,C 180,E1 14255.756,E2 14255.756} C_VEL
LIN {X 0,Y 299.024,Z 1175.132,A -85,B 0,C 180,E1 14251.123,E2 14251.123} C_VEL
LIN {X 0,Y 289.335,Z 1181.792,A -85,B 0,C 180,E1 14246.258,E2 14246.258} C_VEL
LIN {X 0,Y 282.592,Z 1186.08,A -85,B 0,C 180,E1 14241.595,E2 14241.595} C_VEL
LIN {X 0,Y 277.565,Z 1188.805,A -85,B 0,C 180,E1 14236.538,E2 14236.538} C_VEL
LIN {X 0,Y 274.605,Z 1189.686,A -85,B 0,C 180,E1 14231.77,E2 14231.77} C_VEL
LIN {X 0,Y 273.09,Z 1188.974,A -85,B 0,C 180,E1 14227.367,E2 14227.367} C_VEL
LIN {X 0,Y 272.4,Z 1186.797,A -85,B 0,C 180,E1 14222.95,E2 14222.95} C_VEL
LIN {X 0,Y 272.207,Z 1183.519,A -85,B 0,C 180,E1 14218.952,E2 14218.952} C_VEL
LIN {X 0,Y 272.231,Z 1178.775,A -85,B 0,C 180,E1 14214.947,E2 14214.947} C_VEL
LIN {X 0,Y 272.569,Z 1172.602,A -85,B 0,C 180,E1 14210.929,E2 14210.929} C_VEL
LIN {X 0,Y 273.405,Z 1164.632,A -85,B 0,C 180,E1 14206.899,E2 14206.899} C_VEL
LIN {X 0,Y 274.92,Z 1154.874,A -85,B 0,C 180,E1 14202.872,E2 14202.872} C_VEL
LIN {X 0,Y 277.109,Z 1143.792,A -85,B 0,C 180,E1 14199.076,E2 14199.076} C_VEL
LIN {X 0,Y 280.107,Z 1130.573,A -85,B 0,C 180,E1 14195.319,E2 14195.319} C_VEL
LIN {X 0,Y 283.718,Z 1115.861,A -85,B 0,C 180,E1 14191.825,E2 14191.825} C_VEL
LIN {X 0,Y 287.981,Z 1099.174,A -85,B 0,C 180,E1 14188.503,E2 14188.503} C_VEL
LIN {X 0,Y 292.757,Z 1080.488,A -85,B 0,C 180,E1 14185.401,E2 14185.401} C_VEL
LIN {X 0,Y 297.459,Z 1061.511,A -85,B 0,C 180,E1 14182.773,E2 14182.773} C_VEL
LIN {X 0,Y 302.189,Z 1041.368,A -85,B 0,C 180,E1 14180.443,E2 14180.443} C_VEL
LIN {X 0,Y 307.061,Z 1018.757,A -85,B 0,C 180,E1 14178.295,E2 14178.295} C_VEL
LIN {X 0,Y 311.576,Z 995.17,A -85,B 0,C 180,E1 14176.493,E2 14176.493} C_VEL
LIN {X 0,Y 315.511,Z 971.035,A -85,B 0,C 180,E1 14175.039,E2 14175.039} C_VEL
LIN {X 0,Y 318.761,Z 946.631,A -85,B 0,C 180,E1 14173.921,E2 14173.921} C_VEL
LIN {X 0,Y 323.649,Z 899.067,A -85,B 0,C 180,E1 14172.364,E2 14172.364} C_VEL
LIN {X 0,Y 337.153,Z 770.545,A -85,B 0,C 180,E1 14168.474,E2 14168.474} C_VEL
LIN {X 0,Y 321.659,Z 742.247,A -85,B 0,C 180,E1 14165.135,E2 14165.135} C_VEL
LIN {X 0,Y 306.666,Z 716.202,A -85,B 0,C 180,E1 14161.53,E2 14161.53} C_VEL
LIN {X 0,Y 293.313,Z 694.47,A -85,B 0,C 180,E1 14158.015,E2 14158.015} C_VEL
LIN {X 0,Y 284.231,Z 680.523,A -85,B 0,C 180,E1 14155.418,E2 14155.418} C_VEL
LIN {X 0,Y 281.247,Z 676.022,A -85,B 0,C 180,E1 14154.526,E2 14154.526} C_VEL
LIN {X 0,Y 278.85,Z 672.012,A -85,B 0,C 180,E1 14153.765,E2 14153.765} C_VEL
LIN {X 0,Y 276.201,Z 668.563,A -85,B 0,C 180,E1 14152.962,E2 14152.962} C_VEL
LIN {X 0,Y 275.577,Z 666.331,A -85,B 0,C 180,E1 14152.622,E2 14152.622} C_VEL
LIN {X 0,Y 275.621,Z 666.321,A -85,B 0,C 180,E1 14147.745,E2 14147.745} C_VEL
LIN {X 0,Y 275.641,Z 666.314,A -85,B 0,C 180,E1 14143.213,E2 14143.213} C_VEL
LIN {X 0,Y 275.622,Z 666.314,A -85,B 0,C 180,E1 14138.557,E2 14138.557} C_VEL
LIN {X 0,Y 275.574,Z 666.324,A -85,B 0,C 180,E1 14133.747,E2 14133.747} C_VEL
LIN {X 0,Y 275.632,Z 666.334,A -85,B 0,C 180,E1 14128.964,E2 14128.964} C_VEL
LIN {X 0,Y 275.639,Z 666.321,A -85,B 0,C 180,E1 14124.173,E2 14124.173} C_VEL
LIN {X 0,Y 275.602,Z 666.305,A -85,B 0,C 180,E1 14119.449,E2 14119.449} C_VEL
LIN {X 0,Y 275.606,Z 666.339,A -85,B 0,C 180,E1 14114.646,E2 14114.646} C_VEL
LIN {X 0,Y 275.622,Z 666.331,A -85,B 0,C 180,E1 14109.844,E2 14109.844} C_VEL
LIN {X 0,Y 275.636,Z 666.334,A -85,B 0,C 180,E1 14105.119,E2 14105.119} C_VEL
LIN {X 0,Y 275.606,Z 666.353,A -85,B 0,C 180,E1 14100.916,E2 14100.916} C_VEL
LIN {X 0,Y 284.724,Z 691.658,A -85,B 0,C 180,E1 14096.544,E2 14096.544} C_VEL
LIN {X 0,Y 291.689,Z 713.205,A -85,B 0,C 180,E1 14093.142,E2 14093.142} C_VEL
LIN {X 0,Y 298.203,Z 736.668,A -85,B 0,C 180,E1 14089.678,E2 14089.678} C_VEL
LIN {X 0,Y 294.529,Z 774.912,A -85,B 0,C 180,E1 14085.466,E2 14085.466} C_VEL
LIN {X 0,Y 290.413,Z 819.11,A -85,B 0,C 180,E1 14080.59,E2 14080.59} C_VEL
LIN {X 0,Y 287.462,Z 852.826,A -85,B 0,C 180,E1 14076.874,E2 14076.874} C_VEL
LIN {X 0,Y 286.382,Z 859.987,A -85,B 0,C 180,E1 14076.162,E2 14076.162} C_VEL
LIN {X 0,Y 280.959,Z 985.62,A -85,B 0,C 180,E1 14071.515,E2 14071.515} C_VEL
LIN {X 0,Y 280.369,Z 1009.576,A -85,B 0,C 180,E1 14070.509,E2 14070.509} C_VEL
LIN {X 0,Y 279.637,Z 1026.457,A -85,B 0,C 180,E1 14069.444,E2 14069.444} C_VEL
LIN {X 0,Y 278.633,Z 1044.053,A -85,B 0,C 180,E1 14067.91,E2 14067.91} C_VEL
LIN {X 0,Y 277.506,Z 1060.037,A -85,B 0,C 180,E1 14066.072,E2 14066.072} C_VEL
LIN {X 0,Y 276.431,Z 1074.192,A -85,B 0,C 180,E1 14064.007,E2 14064.007} C_VEL
LIN {X 0,Y 275.45,Z 1087.07,A -85,B 0,C 180,E1 14061.686,E2 14061.686} C_VEL
LIN {X 0,Y 274.679,Z 1098.542,A -85,B 0,C 180,E1 14059.119,E2 14059.119} C_VEL
LIN {X 0,Y 274.185,Z 1108.747,A -85,B 0,C 180,E1 14056.303,E2 14056.303} C_VEL
LIN {X 0,Y 274.034,Z 1117.927,A -85,B 0,C 180,E1 14053.054,E2 14053.054} C_VEL
LIN {X 0,Y 274.04,Z 1118.415,A -85,B 0,C 180,E1 14052.86,E2 14052.86} C_VEL
LIN {X 0,Y 273.143,Z 1121.826,A -85,B 0,C 180,E1 14051.411,E2 14051.411} C_VEL
LIN {X 0,Y 269.292,Z 1126.852,A -85,B 0,C 180,E1 14048.771,E2 14048.771} C_VEL
LIN {X 0,Y 267.416,Z 1129.805,A -85,B 0,C 180,E1 14046.754,E2 14046.754} C_VEL
LIN {X 0,Y 267.439,Z 1130.828,A -85,B 0,C 180,E1 14045.947,E2 14045.947} C_VEL
LIN {X 0,Y 269.13,Z 1133.968,A -85,B 0,C 180,E1 14042.551,E2 14042.551} C_VEL
LIN {X 0,Y 271.631,Z 1135.329,A -85,B 0,C 180,E1 14039.152,E2 14039.152} C_VEL
LIN {X 0,Y 274.936,Z 1134.76,A -85,B 0,C 180,E1 14035.824,E2 14035.824} C_VEL
LIN {X 0,Y 279.065,Z 1132.364,A -85,B 0,C 180,E1 14032.585,E2 14032.585} C_VEL
LIN {X 0,Y 283.644,Z 1128.278,A -85,B 0,C 180,E1 14029.639,E2 14029.639} C_VEL
LIN {X 0,Y 288.888,Z 1122.375,A -85,B 0,C 180,E1 14026.791,E2 14026.791} C_VEL
LIN {X 0,Y 294.325,Z 1114.994,A -85,B 0,C 180,E1 14024.226,E2 14024.226} C_VEL
LIN {X 0,Y 300.263,Z 1105.542,A -85,B 0,C 180,E1 14021.754,E2 14021.754} C_VEL
LIN {X 0,Y 306.145,Z 1094.451,A -85,B 0,C 180,E1 14019.541,E2 14019.541} C_VEL
LIN {X 0,Y 311.619,Z 1082.385,A -85,B 0,C 180,E1 14017.648,E2 14017.648} C_VEL
LIN {X 0,Y 317.083,Z 1068.038,A -85,B 0,C 180,E1 14015.894,E2 14015.894} C_VEL
LIN {X 0,Y 321.389,Z 1053.975,A -85,B 0,C 180,E1 14014.571,E2 14014.571} C_VEL
LIN {X 0,Y 324.7,Z 1040.718,A -85,B 0,C 180,E1 14013.574,E2 14013.574} C_VEL
LIN {X 0,Y 327.644,Z 1025.577,A -85,B 0,C 180,E1 14012.68,E2 14012.68} C_VEL
LIN {X 0,Y 332.682,Z 992.101,A -85,B 0,C 180,E1 14011.284,E2 14011.284} C_VEL
LIN {X 0,Y 349.89,Z 892.793,A -85,B 0,C 180,E1 14007.96,E2 14007.96} C_VEL
LIN {X 0,Y 350.695,Z 884.793,A -85,B 0,C 180,E1 14007.196,E2 14007.196} C_VEL
LIN {X 0,Y 360.085,Z 857.085,A -85,B 0,C 180,E1 14004.13,E2 14004.13} C_VEL
LIN {X 0,Y 357.296,Z 863.151,A -85,B 0,C 180,E1 14003.805,E2 14003.805} C_VEL
LIN {X 0,Y 350.782,Z 877.599,A -85,B 0,C 180,E1 14003.083,E2 14003.083} C_VEL
LIN {X 0,Y 347.983,Z 884.089,A -85,B 0,C 180,E1 14002.738,E2 14002.738} C_VEL
LIN {X 0,Y 344.674,Z 892.889,A -85,B 0,C 180,E1 14002.313,E2 14002.313} C_VEL
LIN {X 0,Y 342.108,Z 903.593,A -85,B 0,C 180,E1 14001.718,E2 14001.718} C_VEL
LIN {X 0,Y 334.34,Z 937.815,A -85,B 0,C 180,E1 14000.422,E2 14000.422} C_VEL
LIN {X 0,Y 330.445,Z 955.387,A -85,B 0,C 180,E1 13999.624,E2 13999.624} C_VEL
LIN {X 0,Y 323.895,Z 985.738,A -85,B 0,C 180,E1 13998.416,E2 13998.416} C_VEL
LIN {X 0,Y 316.745,Z 1021.708,A -85,B 0,C 180,E1 13996.585,E2 13996.585} C_VEL
LIN {X 0,Y 311.71,Z 1049.235,A -85,B 0,C 180,E1 13994.865,E2 13994.865} C_VEL
LIN {X 0,Y 306.495,Z 1070.664,A -85,B 0,C 180,E1 13993.11,E2 13993.11} C_VEL
LIN {X 0,Y 302.331,Z 1084.514,A -85,B 0,C 180,E1 13991.787,E2 13991.787} C_VEL
LIN {X 0,Y 297.197,Z 1099.657,A -85,B 0,C 180,E1 13989.982,E2 13989.982} C_VEL
LIN {X 0,Y 290.865,Z 1116.693,A -85,B 0,C 180,E1 13987.425,E2 13987.425} C_VEL
LIN {X 0,Y 284.914,Z 1131.478,A -85,B 0,C 180,E1 13984.644,E2 13984.644} C_VEL
LIN {X 0,Y 279.348,Z 1144.897,A -85,B 0,C 180,E1 13981.502,E2 13981.502} C_VEL
LIN {X 0,Y 274.446,Z 1156.713,A -85,B 0,C 180,E1 13978.03,E2 13978.03} C_VEL
LIN {X 0,Y 270.563,Z 1166.356,A -85,B 0,C 180,E1 13974.447,E2 13974.447} C_VEL
LIN {X 0,Y 267.673,Z 1174.484,A -85,B 0,C 180,E1 13970.553,E2 13970.553} C_VEL
LIN {X 0,Y 266.631,Z 1178.251,A -85,B 0,C 180,E1 13968.358,E2 13968.358} C_VEL
LIN {X 0,Y 265.344,Z 1187.785,A -85,B 0,C 180,E1 13964.398,E2 13964.398} C_VEL
LIN {X 0,Y 264.742,Z 1195.936,A -85,B 0,C 180,E1 13960.222,E2 13960.222} C_VEL
LIN {X 0,Y 264.663,Z 1201.967,A -85,B 0,C 180,E1 13956.287,E2 13956.287} C_VEL
LIN {X 0,Y 264.725,Z 1206.309,A -85,B 0,C 180,E1 13952.378,E2 13952.378} C_VEL
LIN {X 0,Y 264.604,Z 1208.95,A -85,B 0,C 180,E1 13948.914,E2 13948.914} C_VEL
LIN {X 0,Y 264.253,Z 1210.692,A -85,B 0,C 180,E1 13944.787,E2 13944.787} C_VEL
LIN {X 0,Y 264.211,Z 1210.957,A -85,B 0,C 180,E1 13940.412,E2 13940.412} C_VEL
LIN {X 0,Y 265.221,Z 1209.604,A -85,B 0,C 180,E1 13935.366,E2 13935.366} C_VEL
LIN {X 0,Y 267.841,Z 1206.55,A -85,B 0,C 180,E1 13930.365,E2 13930.365} C_VEL
LIN {X 0,Y 272.795,Z 1201.377,A -85,B 0,C 180,E1 13925.067,E2 13925.067} C_VEL
LIN {X 0,Y 280.768,Z 1193.849,A -85,B 0,C 180,E1 13919.62,E2 13919.62} C_VEL
LIN {X 0,Y 291.032,Z 1184.801,A -85,B 0,C 180,E1 13914.744,E2 13914.744} C_VEL
LIN {X 0,Y 304.299,Z 1173.653,A -85,B 0,C 180,E1 13910.15,E2 13910.15} C_VEL
LIN {X 0,Y 320.077,Z 1160.845,A -85,B 0,C 180,E1 13906.089,E2 13906.089} C_VEL
LIN {X 0,Y 333.238,Z 1150.539,A -85,B 0,C 180,E1 13903.438,E2 13903.438} C_VEL
LIN {X 0,Y 316.373,Z 1161.782,A -85,B 0,C 180,E1 13899.678,E2 13899.678} C_VEL
LIN {X 0,Y 301.359,Z 1171.586,A -85,B 0,C 180,E1 13895.266,E2 13895.266} C_VEL
LIN {X 0,Y 289.31,Z 1179.195,A -85,B 0,C 180,E1 13890.538,E2 13890.538} C_VEL
LIN {X 0,Y 280.343,Z 1184.517,A -85,B 0,C 180,E1 13885.798,E2 13885.798} C_VEL
LIN {X 0,Y 273.51,Z 1188.158,A -85,B 0,C 180,E1 13880.774,E2 13880.774} C_VEL
LIN {X 0,Y 268.927,Z 1190.009,A -85,B 0,C 180,E1 13875.753,E2 13875.753} C_VEL
LIN {X 0,Y 266.186,Z 1190.138,A -85,B 0,C 180,E1 13870.83,E2 13870.83} C_VEL
LIN {X 0,Y 264.818,Z 1188.637,A -85,B 0,C 180,E1 13866.073,E2 13866.073} C_VEL
LIN {X 0,Y 264.306,Z 1185.759,A -85,B 0,C 180,E1 13861.522,E2 13861.522} C_VEL
LIN {X 0,Y 264.184,Z 1181.943,A -85,B 0,C 180,E1 13857.619,E2 13857.619} C_VEL
LIN {X 0,Y 264.325,Z 1176.239,A -85,B 0,C 180,E1 13853.27,E2 13853.27} C_VEL
LIN {X 0,Y 264.822,Z 1169.572,A -85,B 0,C 180,E1 13849.343,E2 13849.343} C_VEL
LIN {X 0,Y 265.94,Z 1160.816,A -85,B 0,C 180,E1 13845.192,E2 13845.192} C_VEL
LIN {X 0,Y 267.817,Z 1150.17,A -85,B 0,C 180,E1 13841.051,E2 13841.051} C_VEL
LIN {X 0,Y 270.42,Z 1138.103,A -85,B 0,C 180,E1 13837.16,E2 13837.16} C_VEL
LIN {X 0,Y 273.676,Z 1124.553,A -85,B 0,C 180,E1 13833.528,E2 13833.528} C_VEL
LIN {X 0,Y 277.722,Z 1108.786,A -85,B 0,C 180,E1 13829.976,E2 13829.976} C_VEL
LIN {X 0,Y 282.284,Z 1091.42,A -85,B 0,C 180,E1 13826.706,E2 13826.706} C_VEL
LIN {X 0,Y 287.033,Z 1073.096,A -85,B 0,C 180,E1 13823.817,E2 13823.817} C_VEL
LIN {X 0,Y 291.992,Z 1053.216,A -85,B 0,C 180,E1 13821.202,E2 13821.202} C_VEL
LIN {X 0,Y 297.014,Z 1031.488,A -85,B 0,C 180,E1 13818.848,E2 13818.848} C_VEL
LIN {X 0,Y 301.812,Z 1008.619,A -85,B 0,C 180,E1 13816.84,E2 13816.84} C_VEL
LIN {X 0,Y 305.99,Z 985.844,A -85,B 0,C 180,E1 13815.234,E2 13815.234} C_VEL
LIN {X 0,Y 309.698,Z 962.062,A -85,B 0,C 180,E1 13813.913,E2 13813.913} C_VEL
LIN {X 0,Y 312.779,Z 937.725,A -85,B 0,C 180,E1 13812.897,E2 13812.897} C_VEL
LIN {X 0,Y 330.419,Z 773.314,A -85,B 0,C 180,E1 13807.741,E2 13807.741} C_VEL
LIN {X 0,Y 314.403,Z 743.937,A -85,B 0,C 180,E1 13804.149,E2 13804.149} C_VEL
LIN {X 0,Y 299.197,Z 717.653,A -85,B 0,C 180,E1 13800.365,E2 13800.365} C_VEL
LIN {X 0,Y 286.004,Z 696.178,A -85,B 0,C 180,E1 13796.726,E2 13796.726} C_VEL
LIN {X 0,Y 276.65,Z 681.954,A -85,B 0,C 180,E1 13793.938,E2 13793.938} C_VEL
LIN {X 0,Y 273.316,Z 676.958,A -85,B 0,C 180,E1 13792.876,E2 13792.876} C_VEL
LIN {X 0,Y 270.473,Z 672.481,A -85,B 0,C 180,E1 13791.927,E2 13791.927} C_VEL
LIN {X 0,Y 268.228,Z 669.468,A -85,B 0,C 180,E1 13791.201,E2 13791.201} C_VEL
LIN {X 0,Y 267.64,Z 667.327,A -85,B 0,C 180,E1 13790.906,E2 13790.906} C_VEL
LIN {X 0,Y 267.692,Z 667.324,A -85,B 0,C 180,E1 13786.049,E2 13786.049} C_VEL
LIN {X 0,Y 267.7,Z 667.323,A -85,B 0,C 180,E1 13781.421,E2 13781.421} C_VEL
LIN {X 0,Y 267.672,Z 667.319,A -85,B 0,C 180,E1 13776.653,E2 13776.653} C_VEL
LIN {X 0,Y 267.653,Z 667.308,A -85,B 0,C 180,E1 13771.501,E2 13771.501} C_VEL
LIN {X 0,Y 267.694,Z 667.297,A -85,B 0,C 180,E1 13767.005,E2 13767.005} C_VEL
LIN {X 0,Y 267.707,Z 667.323,A -85,B 0,C 180,E1 13762.276,E2 13762.276} C_VEL
LIN {X 0,Y 267.644,Z 667.301,A -85,B 0,C 180,E1 13757.489,E2 13757.489} C_VEL
LIN {X 0,Y 267.677,Z 667.319,A -85,B 0,C 180,E1 13752.616,E2 13752.616} C_VEL
LIN {X 0,Y 267.697,Z 667.324,A -85,B 0,C 180,E1 13747.84,E2 13747.84} C_VEL
LIN {X 0,Y 267.686,Z 667.324,A -85,B 0,C 180,E1 13743.133,E2 13743.133} C_VEL
LIN {X 0,Y 267.725,Z 667.572,A -85,B 0,C 180,E1 13741.75,E2 13741.75} C_VEL
LIN {X 0,Y 275.854,Z 689.758,A -85,B 0,C 180,E1 13737.807,E2 13737.807} C_VEL
LIN {X 0,Y 283.271,Z 712.172,A -85,B 0,C 180,E1 13734.134,E2 13734.134} C_VEL
LIN {X 0,Y 289.311,Z 733.396,A -85,B 0,C 180,E1 13730.9,E2 13730.9} C_VEL
LIN {X 0,Y 290.745,Z 739.116,A -85,B 0,C 180,E1 13730.069,E2 13730.069} C_VEL
LIN {X 0,Y 286.357,Z 782.38,A -85,B 0,C 180,E1 13725.229,E2 13725.229} C_VEL
LIN {X 0,Y 282.188,Z 826.071,A -85,B 0,C 180,E1 13720.323,E2 13720.323} C_VEL
LIN {X 0,Y 279.551,Z 854.121,A -85,B 0,C 180,E1 13717.185,E2 13717.185} C_VEL
LIN {X 0,Y 278.572,Z 860.777,A -85,B 0,C 180,E1 13716.522,E2 13716.522} C_VEL
LIN {X 0,Y 273.031,Z 985.731,A -85,B 0,C 180,E1 13711.736,E2 13711.736} C_VEL
LIN {X 0,Y 272.409,Z 1010.08,A -85,B 0,C 180,E1 13710.681,E2 13710.681} C_VEL
LIN {X 0,Y 271.634,Z 1027.403,A -85,B 0,C 180,E1 13709.549,E2 13709.549} C_VEL
LIN {X 0,Y 270.614,Z 1044.786,A -85,B 0,C 180,E1 13707.98,E2 13707.98} C_VEL
LIN {X 0,Y 269.489,Z 1060.446,A -85,B 0,C 180,E1 13706.126,E2 13706.126} C_VEL
LIN {X 0,Y 268.435,Z 1074.227,A -85,B 0,C 180,E1 13704.088,E2 13704.088} C_VEL
LIN {X 0,Y 267.36,Z 1088.292,A -85,B 0,C 180,E1 13701.495,E2 13701.495} C_VEL
LIN {X 0,Y 266.601,Z 1099.907,A -85,B 0,C 180,E1 13698.811,E2 13698.811} C_VEL
LIN {X 0,Y 266.142,Z 1110.04,A -85,B 0,C 180,E1 13695.913,E2 13695.913} C_VEL
LIN {X 0,Y 266.049,Z 1119.086,A -85,B 0,C 180,E1 13692.585,E2 13692.585} C_VEL
LIN {X 0,Y 266.413,Z 1125.484,A -85,B 0,C 180,E1 13689.5,E2 13689.5} C_VEL
LIN {X 0,Y 267.439,Z 1130.828,A -85,B 0,C 180,E1 13685.947,E2 13685.947} C_VEL
LIN {X 0,Y 267.157,Z 1132.663,A -85,B 0,C 180,E1 13684.33,E2 13684.33} C_VEL
LIN {X 0,Y 264.212,Z 1135.454,A -85,B 0,C 180,E1 13680.94,E2 13680.94} C_VEL
LIN {X 0,Y 263.826,Z 1136.347,A -85,B 0,C 180,E1 13679.018,E2 13679.018} C_VEL
LIN {X 0,Y 264.213,Z 1136.483,A -85,B 0,C 180,E1 13678.422,E2 13678.422} C_VEL
LIN {X 0,Y 267.719,Z 1136.081,A -85,B 0,C 180,E1 13675.068,E2 13675.068} C_VEL
LIN {X 0,Y 272.122,Z 1133.82,A -85,B 0,C 180,E1 13671.757,E2 13671.757} C_VEL
LIN {X 0,Y 277.002,Z 1129.946,A -85,B 0,C 180,E1 13668.755,E2 13668.755} C_VEL
LIN {X 0,Y 282.951,Z 1123.781,A -85,B 0,C 180,E1 13665.674,E2 13665.674} C_VEL
LIN {X 0,Y 288.733,Z 1116.491,A -85,B 0,C 180,E1 13663.084,E2 13663.084} C_VEL
LIN {X 0,Y 295.023,Z 1107.139,A -85,B 0,C 180,E1 13660.597,E2 13660.597} C_VEL
LIN {X 0,Y 300.887,Z 1096.885,A -85,B 0,C 180,E1 13658.5,E2 13658.5} C_VEL
LIN {X 0,Y 307.032,Z 1084.35,A -85,B 0,C 180,E1 13656.484,E2 13656.484} C_VEL
LIN {X 0,Y 313.053,Z 1069.526,A -85,B 0,C 180,E1 13654.656,E2 13654.656} C_VEL
LIN {X 0,Y 317.595,Z 1055.616,A -85,B 0,C 180,E1 13653.34,E2 13653.34} C_VEL
LIN {X 0,Y 321.09,Z 1042.577,A -85,B 0,C 180,E1 13652.351,E2 13652.351} C_VEL
LIN {X 0,Y 324.264,Z 1027.397,A -85,B 0,C 180,E1 13651.445,E2 13651.445} C_VEL
LIN {X 0,Y 329.541,Z 994.608,A -85,B 0,C 180,E1 13650.061,E2 13650.061} C_VEL
LIN {X 0,Y 347.594,Z 895.179,A -85,B 0,C 180,E1 13646.743,E2 13646.743} C_VEL
LIN {X 0,Y 348.916,Z 885.846,A -85,B 0,C 180,E1 13645.825,E2 13645.825} C_VEL
LIN {X 0,Y 352.626,Z 875.085,A -85,B 0,C 180,E1 13644.604,E2 13644.604} C_VEL
LIN {X 0,Y 347.779,Z 885.772,A -85,B 0,C 180,E1 13644.026,E2 13644.026} C_VEL
LIN {X 0,Y 345.645,Z 891.476,A -85,B 0,C 180,E1 13643.773,E2 13643.773} C_VEL
LIN {X 0,Y 341.932,Z 905.93,A -85,B 0,C 180,E1 13643.008,E2 13643.008} C_VEL
LIN {X 0,Y 333.722,Z 940.563,A -85,B 0,C 180,E1 13641.715,E2 13641.715} C_VEL
LIN {X 0,Y 329.833,Z 957.2,A -85,B 0,C 180,E1 13640.974,E2 13640.974} C_VEL
LIN {X 0,Y 322.925,Z 987.673,A -85,B 0,C 180,E1 13639.781,E2 13639.781} C_VEL
LIN {X 0,Y 315.259,Z 1023.722,A -85,B 0,C 180,E1 13637.963,E2 13637.963} C_VEL
LIN {X 0,Y 309.989,Z 1049.348,A -85,B 0,C 180,E1 13636.376,E2 13636.376} C_VEL
LIN {X 0,Y 304.597,Z 1069.162,A -85,B 0,C 180,E1 13634.755,E2 13634.755} C_VEL
LIN {X 0,Y 299.467,Z 1084.53,A -85,B 0,C 180,E1 13633.321,E2 13633.321} C_VEL
LIN {X 0,Y 293.082,Z 1101.153,A -85,B 0,C 180,E1 13631.307,E2 13631.307} C_VEL
LIN {X 0,Y 286.426,Z 1116.965,A -85,B 0,C 180,E1 13628.873,E2 13628.873} C_VEL
LIN {X 0,Y 279.508,Z 1132.241,A -85,B 0,C 180,E1 13625.918,E2 13625.918} C_VEL
LIN {X 0,Y 273.046,Z 1145.844,A -85,B 0,C 180,E1 13622.565,E2 13622.565} C_VEL
LIN {X 0,Y 267.957,Z 1156.52,A -85,B 0,C 180,E1 13619.26,E2 13619.26} C_VEL
LIN {X 0,Y 263.397,Z 1166.39,A -85,B 0,C 180,E1 13615.372,E2 13615.372} C_VEL
LIN {X 0,Y 260.284,Z 1173.757,A -85,B 0,C 180,E1 13611.61,E2 13611.61} C_VEL
LIN {X 0,Y 258.325,Z 1179.661,A -85,B 0,C 180,E1 13607.569,E2 13607.569} C_VEL
LIN {X 0,Y 257.189,Z 1188.937,A -85,B 0,C 180,E1 13603.486,E2 13603.486} C_VEL
LIN {X 0,Y 256.752,Z 1196.308,A -85,B 0,C 180,E1 13599.411,E2 13599.411} C_VEL
LIN {X 0,Y 256.748,Z 1202.103,A -85,B 0,C 180,E1 13595.36,E2 13595.36} C_VEL
LIN {X 0,Y 256.783,Z 1206.029,A -85,B 0,C 180,E1 13591.559,E2 13591.559} C_VEL
LIN {X 0,Y 256.583,Z 1208.554,A -85,B 0,C 180,E1 13587.987,E2 13587.987} C_VEL
LIN {X 0,Y 256.215,Z 1210.192,A -85,B 0,C 180,E1 13583.499,E2 13583.499} C_VEL
LIN {X 0,Y 256.361,Z 1210.335,A -85,B 0,C 180,E1 13578.979,E2 13578.979} C_VEL
LIN {X 0,Y 257.925,Z 1208.735,A -85,B 0,C 180,E1 13573.558,E2 13573.558} C_VEL
LIN {X 0,Y 261.427,Z 1205.427,A -85,B 0,C 180,E1 13568.22,E2 13568.22} C_VEL
LIN {X 0,Y 267.366,Z 1200.123,A -85,B 0,C 180,E1 13562.852,E2 13562.852} C_VEL
LIN {X 0,Y 276.363,Z 1192.662,A -85,B 0,C 180,E1 13557.465,E2 13557.465} C_VEL
LIN {X 0,Y 287.929,Z 1183.602,A -85,B 0,C 180,E1 13552.572,E2 13552.572} C_VEL
LIN {X 0,Y 302.971,Z 1172.275,A -85,B 0,C 180,E1 13547.934,E2 13547.934} C_VEL
LIN {X 0,Y 319.99,Z 1159.774,A -85,B 0,C 180,E1 13544.051,E2 13544.051} C_VEL
LIN {X 0,Y 323.345,Z 1157.401,A -85,B 0,C 180,E1 13543.358,E2 13543.358} C_VEL
LIN {X 0,Y 306.046,Z 1167.776,A -85,B 0,C 180,E1 13539.337,E2 13539.337} C_VEL
LIN {X 0,Y 291.702,Z 1176.093,A -85,B 0,C 180,E1 13534.925,E2 13534.925} C_VEL
LIN {X 0,Y 280.188,Z 1182.448,A -85,B 0,C 180,E1 13530.215,E2 13530.215} C_VEL
LIN {X 0,Y 271.027,Z 1187.1,A -85,B 0,C 180,E1 13525.109,E2 13525.109} C_VEL
LIN {X 0,Y 264.461,Z 1189.883,A -85,B 0,C 180,E1 13519.898,E2 13519.898} C_VEL
LIN {X 0,Y 260.168,Z 1190.913,A -85,B 0,C 180,E1 13514.698,E2 13514.698} C_VEL
LIN {X 0,Y 257.713,Z 1190.176,A -85,B 0,C 180,E1 13509.608,E2 13509.608} C_VEL
LIN {X 0,Y 256.562,Z 1187.804,A -85,B 0,C 180,E1 13504.475,E2 13504.475} C_VEL
LIN {X 0,Y 256.235,Z 1184.312,A -85,B 0,C 180,E1 13500.005,E2 13500.005} C_VEL
LIN {X 0,Y 256.206,Z 1179.487,A -85,B 0,C 180,E1 13495.753,E2 13495.753} C_VEL
LIN {X 0,Y 256.504,Z 1173.256,A -85,B 0,C 180,E1 13491.487,E2 13491.487} C_VEL
LIN {X 0,Y 257.299,Z 1165.242,A -85,B 0,C 180,E1 13487.208,E2 13487.208} C_VEL
LIN {X 0,Y 258.82,Z 1155.419,A -85,B 0,C 180,E1 13482.931,E2 13482.931} C_VEL
LIN {X 0,Y 261.064,Z 1144.283,A -85,B 0,C 180,E1 13478.904,E2 13478.904} C_VEL
LIN {X 0,Y 264.181,Z 1131.006,A -85,B 0,C 180,E1 13474.924,E2 13474.924} C_VEL
LIN {X 0,Y 267.954,Z 1116.21,A -85,B 0,C 180,E1 13471.231,E2 13471.231} C_VEL
LIN {X 0,Y 272.427,Z 1099.454,A -85,B 0,C 180,E1 13467.728,E2 13467.728} C_VEL
LIN {X 0,Y 277.346,Z 1081.069,A -85,B 0,C 180,E1 13464.525,E2 13464.525} C_VEL
LIN {X 0,Y 282.379,Z 1061.651,A -85,B 0,C 180,E1 13461.715,E2 13461.715} C_VEL
LIN {X 0,Y 287.347,Z 1041.421,A -85,B 0,C 180,E1 13459.28,E2 13459.28} C_VEL
LIN {X 0,Y 292.307,Z 1019.482,A -85,B 0,C 180,E1 13457.107,E2 13457.107} C_VEL
LIN {X 0,Y 296.922,Z 996.541,A -85,B 0,C 180,E1 13455.274,E2 13455.274} C_VEL
LIN {X 0,Y 301.01,Z 972.932,A -85,B 0,C 180,E1 13453.776,E2 13453.776} C_VEL
LIN {X 0,Y 304.434,Z 948.962,A -85,B 0,C 180,E1 13452.602,E2 13452.602} C_VEL
LIN {X 0,Y 308.48,Z 912.852,A -85,B 0,C 180,E1 13451.323,E2 13451.323} C_VEL
LIN {X 0,Y 323.638,Z 775.977,A -85,B 0,C 180,E1 13446.965,E2 13446.965} C_VEL
LIN {X 0,Y 308.31,Z 747.799,A -85,B 0,C 180,E1 13443.433,E2 13443.433} C_VEL
LIN {X 0,Y 293.725,Z 722.469,A -85,B 0,C 180,E1 13439.692,E2 13439.692} C_VEL
LIN {X 0,Y 281.271,Z 701.988,A -85,B 0,C 180,E1 13436.158,E2 13436.158} C_VEL
LIN {X 0,Y 271.63,Z 687.271,A -85,B 0,C 180,E1 13433.199,E2 13433.199} C_VEL
LIN {X 0,Y 265.699,Z 678.323,A -85,B 0,C 180,E1 13431.239,E2 13431.239} C_VEL
LIN {X 0,Y 263.154,Z 674.233,A -85,B 0,C 180,E1 13430.347,E2 13430.347} C_VEL
LIN {X 0,Y 260.381,Z 670.621,A -85,B 0,C 180,E1 13429.403,E2 13429.403} C_VEL
LIN {X 0,Y 259.719,Z 668.305,A -85,B 0,C 180,E1 13429.046,E2 13429.046} C_VEL
LIN {X 0,Y 259.769,Z 668.291,A -85,B 0,C 180,E1 13424.037,E2 13424.037} C_VEL
LIN {X 0,Y 259.759,Z 668.292,A -85,B 0,C 180,E1 13419.083,E2 13419.083} C_VEL
LIN {X 0,Y 259.701,Z 668.309,A -85,B 0,C 180,E1 13414.375,E2 13414.375} C_VEL
LIN {X 0,Y 259.749,Z 668.315,A -85,B 0,C 180,E1 13409.341,E2 13409.341} C_VEL
LIN {X 0,Y 259.761,Z 668.291,A -85,B 0,C 180,E1 13404.481,E2 13404.481} C_VEL
LIN {X 0,Y 259.73,Z 668.284,A -85,B 0,C 180,E1 13399.803,E2 13399.803} C_VEL
LIN {X 0,Y 259.716,Z 668.318,A -85,B 0,C 180,E1 13394.827,E2 13394.827} C_VEL
LIN {X 0,Y 259.746,Z 668.308,A -85,B 0,C 180,E1 13389.913,E2 13389.913} C_VEL
LIN {X 0,Y 259.759,Z 668.312,A -85,B 0,C 180,E1 13385.196,E2 13385.196} C_VEL
LIN {X 0,Y 259.783,Z 668.565,A -85,B 0,C 180,E1 13382.682,E2 13382.682} C_VEL
LIN {X 0,Y 268.388,Z 691.871,A -85,B 0,C 180,E1 13378.441,E2 13378.441} C_VEL
LIN {X 0,Y 275.57,Z 713.566,A -85,B 0,C 180,E1 13374.77,E2 13374.77} C_VEL
LIN {X 0,Y 281.864,Z 735.509,A -85,B 0,C 180,E1 13371.37,E2 13371.37} C_VEL
LIN {X 0,Y 283.202,Z 741.719,A -85,B 0,C 180,E1 13370.476,E2 13370.476} C_VEL
LIN {X 0,Y 278.656,Z 784.915,A -85,B 0,C 180,E1 13365.559,E2 13365.559} C_VEL
LIN {X 0,Y 274.389,Z 828.407,A -85,B 0,C 180,E1 13360.591,E2 13360.591} C_VEL
LIN {X 0,Y 271.832,Z 854.361,A -85,B 0,C 180,E1 13357.626,E2 13357.626} C_VEL
LIN {X 0,Y 270.74,Z 861.671,A -85,B 0,C 180,E1 13356.873,E2 13356.873} C_VEL
LIN {X 0,Y 265.091,Z 985.653,A -85,B 0,C 180,E1 13351.945,E2 13351.945} C_VEL
LIN {X 0,Y 264.404,Z 1011.271,A -85,B 0,C 180,E1 13350.788,E2 13350.788} C_VEL
LIN {X 0,Y 263.606,Z 1028.576,A -85,B 0,C 180,E1 13349.615,E2 13349.615} C_VEL
LIN {X 0,Y 262.59,Z 1045.473,A -85,B 0,C 180,E1 13348.045,E2 13348.045} C_VEL
LIN {X 0,Y 261.418,Z 1061.555,A -85,B 0,C 180,E1 13346.089,E2 13346.089} C_VEL
LIN {X 0,Y 260.326,Z 1075.682,A -85,B 0,C 180,E1 13343.926,E2 13343.926} C_VEL
LIN {X 0,Y 259.298,Z 1089.162,A -85,B 0,C 180,E1 13341.365,E2 13341.365} C_VEL
LIN {X 0,Y 258.526,Z 1101.17,A -85,B 0,C 180,E1 13338.485,E2 13338.485} C_VEL
LIN {X 0,Y 258.106,Z 1111.202,A -85,B 0,C 180,E1 13335.498,E2 13335.498} C_VEL
LIN {X 0,Y 258.079,Z 1120.261,A -85,B 0,C 180,E1 13332.071,E2 13332.071} C_VEL
LIN {X 0,Y 258.583,Z 1127.042,A -85,B 0,C 180,E1 13328.669,E2 13328.669} C_VEL
LIN {X 0,Y 259.983,Z 1132.639,A -85,B 0,C 180,E1 13324.628,E2 13324.628} C_VEL
LIN {X 0,Y 262.06,Z 1135.555,A -85,B 0,C 180,E1 13321.088,E2 13321.088} C_VEL
LIN {X 0,Y 264.213,Z 1136.483,A -85,B 0,C 180,E1 13318.422,E2 13318.422} C_VEL
LIN {X 0,Y 264.858,Z 1136.782,A -85,B 0,C 180,E1 13316.746,E2 13316.746} C_VEL
LIN {X 0,Y 263.963,Z 1136.555,A -85,B 0,C 180,E1 13313.115,E2 13313.115} C_VEL
LIN {X 0,Y 264.724,Z 1135.668,A -85,B 0,C 180,E1 13311.327,E2 13311.327} C_VEL
LIN {X 0,Y 265.449,Z 1135.191,A -85,B 0,C 180,E1 13310.758,E2 13310.758} C_VEL
LIN {X 0,Y 270.811,Z 1131.334,A -85,B 0,C 180,E1 13307.63,E2 13307.63} C_VEL
LIN {X 0,Y 277.152,Z 1125.251,A -85,B 0,C 180,E1 13304.512,E2 13304.512} C_VEL
LIN {X 0,Y 283.296,Z 1118.074,A -85,B 0,C 180,E1 13301.901,E2 13301.901} C_VEL
LIN {X 0,Y 289.947,Z 1108.842,A -85,B 0,C 180,E1 13299.402,E2 13299.402} C_VEL
LIN {X 0,Y 296.015,Z 1099.034,A -85,B 0,C 180,E1 13297.348,E2 13297.348} C_VEL
LIN {X 0,Y 302.763,Z 1086.173,A -85,B 0,C 180,E1 13295.25,E2 13295.25} C_VEL
LIN {X 0,Y 309.241,Z 1071.224,A -85,B 0,C 180,E1 13293.392,E2 13293.392} C_VEL
LIN {X 0,Y 314.029,Z 1057.532,A -85,B 0,C 180,E1 13292.088,E2 13292.088} C_VEL
LIN {X 0,Y 317.99,Z 1043.63,A -85,B 0,C 180,E1 13291.034,E2 13291.034} C_VEL
LIN {X 0,Y 321.266,Z 1028.917,A -85,B 0,C 180,E1 13290.156,E2 13290.156} C_VEL
LIN {X 0,Y 326.895,Z 996.118,A -85,B 0,C 180,E1 13288.767,E2 13288.767} C_VEL
LIN {X 0,Y 345.601,Z 897.741,A -85,B 0,C 180,E1 13285.514,E2 13285.514} C_VEL
LIN {X 0,Y 346.166,Z 893.297,A -85,B 0,C 180,E1 13285.063,E2 13285.063} C_VEL
LIN {X 0,Y 342.171,Z 908.286,A -85,B 0,C 180,E1 13284.296,E2 13284.296} C_VEL
LIN {X 0,Y 333.523,Z 943.026,A -85,B 0,C 180,E1 13283.025,E2 13283.025} C_VEL
LIN {X 0,Y 329.574,Z 959.103,A -85,B 0,C 180,E1 13282.326,E2 13282.326} C_VEL
LIN {X 0,Y 322.263,Z 989.869,A -85,B 0,C 180,E1 13281.144,E2 13281.144} C_VEL
LIN {X 0,Y 314.121,Z 1025.842,A -85,B 0,C 180,E1 13279.352,E2 13279.352} C_VEL
LIN {X 0,Y 308.776,Z 1049.185,A -85,B 0,C 180,E1 13277.928,E2 13277.928} C_VEL
LIN {X 0,Y 303.309,Z 1067.279,A -85,B 0,C 180,E1 13276.485,E2 13276.485} C_VEL
LIN {X 0,Y 296.888,Z 1084.763,A -85,B 0,C 180,E1 13274.871,E2 13274.871} C_VEL
LIN {X 0,Y 289.729,Z 1101.606,A -85,B 0,C 180,E1 13272.829,E2 13272.829} C_VEL
LIN {X 0,Y 282.329,Z 1117.216,A -85,B 0,C 180,E1 13270.395,E2 13270.395} C_VEL
LIN {X 0,Y 275.082,Z 1131.484,A -85,B 0,C 180,E1 13267.583,E2 13267.583} C_VEL
LIN {X 0,Y 267.991,Z 1144.718,A -85,B 0,C 180,E1 13264.286,E2 13264.286} C_VEL
LIN {X 0,Y 261.953,Z 1155.789,A -85,B 0,C 180,E1 13260.759,E2 13260.759} C_VEL
LIN {X 0,Y 256.858,Z 1165.412,A -85,B 0,C 180,E1 13256.84,E2 13256.84} C_VEL
LIN {X 0,Y 253.238,Z 1172.599,A -85,B 0,C 180,E1 13253.006,E2 13253.006} C_VEL
LIN {X 0,Y 250.666,Z 1178.651,A -85,B 0,C 180,E1 13248.606,E2 13248.606} C_VEL
LIN {X 0,Y 250.135,Z 1180.451,A -85,B 0,C 180,E1 13246.963,E2 13246.963} C_VEL
LIN {X 0,Y 249.089,Z 1189.867,A -85,B 0,C 180,E1 13242.516,E2 13242.516} C_VEL
LIN {X 0,Y 248.789,Z 1196.994,A -85,B 0,C 180,E1 13238.316,E2 13238.316} C_VEL
LIN {X 0,Y 248.838,Z 1202.394,A -85,B 0,C 180,E1 13234.145,E2 13234.145} C_VEL
LIN {X 0,Y 248.83,Z 1205.703,A -85,B 0,C 180,E1 13230.688,E2 13230.688} C_VEL
LIN {X 0,Y 248.544,Z 1208.116,A -85,B 0,C 180,E1 13226.999,E2 13226.999} C_VEL
LIN {X 0,Y 248.215,Z 1209.637,A -85,B 0,C 180,E1 13222.321,E2 13222.321} C_VEL
LIN {X 0,Y 248.628,Z 1209.695,A -85,B 0,C 180,E1 13217.454,E2 13217.454} C_VEL
LIN {X 0,Y 250.729,Z 1207.993,A -85,B 0,C 180,E1 13211.874,E2 13211.874} C_VEL
LIN {X 0,Y 255.17,Z 1204.47,A -85,B 0,C 180,E1 13206.193,E2 13206.193} C_VEL
LIN {X 0,Y 262.398,Z 1198.941,A -85,B 0,C 180,E1 13200.554,E2 13200.554} C_VEL
LIN {X 0,Y 272.743,Z 1191.392,A -85,B 0,C 180,E1 13195.114,E2 13195.114} C_VEL
LIN {X 0,Y 286.423,Z 1181.827,A -85,B 0,C 180,E1 13190.031,E2 13190.031} C_VEL
LIN {X 0,Y 302.886,Z 1170.699,A -85,B 0,C 180,E1 13185.582,E2 13185.582} C_VEL
LIN {X 0,Y 313.474,Z 1163.649,A -85,B 0,C 180,E1 13183.302,E2 13183.302} C_VEL
LIN {X 0,Y 296.244,Z 1172.874,A -85,B 0,C 180,E1 13179.141,E2 13179.141} C_VEL
LIN {X 0,Y 282.001,Z 1180.153,A -85,B 0,C 180,E1 13174.567,E2 13174.567} C_VEL
LIN {X 0,Y 270.252,Z 1185.73,A -85,B 0,C 180,E1 13169.482,E2 13169.482} C_VEL
LIN {X 0,Y 261.111,Z 1189.503,A -85,B 0,C 180,E1 13163.953,E2 13163.953} C_VEL
LIN {X 0,Y 255.013,Z 1191.289,A -85,B 0,C 180,E1 13158.522,E2 13158.522} C_VEL
LIN {X 0,Y 251.196,Z 1191.323,A -85,B 0,C 180,E1 13153.119,E2 13153.119} C_VEL
LIN {X 0,Y 249.238,Z 1189.76,A -85,B 0,C 180,E1 13148.077,E2 13148.077} C_VEL
LIN {X 0,Y 248.423,Z 1186.9,A -85,B 0,C 180,E1 13143.235,E2 13143.235} C_VEL
LIN {X 0,Y 248.209,Z 1182.881,A -85,B 0,C 180,E1 13138.851,E2 13138.851} C_VEL
LIN {X 0,Y 248.262,Z 1177.526,A -85,B 0,C 180,E1 13134.458,E2 13134.458} C_VEL
LIN {X 0,Y 248.666,Z 1170.935,A -85,B 0,C 180,E1 13130.282,E2 13130.282} C_VEL
LIN {X 0,Y 249.753,Z 1161.813,A -85,B 0,C 180,E1 13125.633,E2 13125.633} C_VEL
LIN {X 0,Y 251.492,Z 1151.851,A -85,B 0,C 180,E1 13121.46,E2 13121.46} C_VEL
LIN {X 0,Y 254.088,Z 1139.856,A -85,B 0,C 180,E1 13117.322,E2 13117.322} C_VEL
LIN {X 0,Y 257.384,Z 1126.532,A -85,B 0,C 180,E1 13113.47,E2 13113.47} C_VEL
LIN {X 0,Y 261.665,Z 1110.474,A -85,B 0,C 180,E1 13109.587,E2 13109.587} C_VEL
LIN {X 0,Y 266.219,Z 1093.86,A -85,B 0,C 180,E1 13106.236,E2 13106.236} C_VEL
LIN {X 0,Y 271.31,Z 1075.145,A -85,B 0,C 180,E1 13103.085,E2 13103.085} C_VEL
LIN {X 0,Y 276.666,Z 1054.674,A -85,B 0,C 180,E1 13100.238,E2 13100.238} C_VEL
LIN {X 0,Y 281.906,Z 1033.102,A -85,B 0,C 180,E1 13097.775,E2 13097.775} C_VEL
LIN {X 0,Y 286.678,Z 1011.661,A -85,B 0,C 180,E1 13095.775,E2 13095.775} C_VEL
LIN {X 0,Y 291.136,Z 989.018,A -85,B 0,C 180,E1 13094.064,E2 13094.064} C_VEL
LIN {X 0,Y 295.241,Z 964.413,A -85,B 0,C 180,E1 13092.6,E2 13092.6} C_VEL
LIN {X 0,Y 298.673,Z 939.194,A -85,B 0,C 180,E1 13091.48,E2 13091.48} C_VEL
LIN {X 0,Y 316.982,Z 778.913,A -85,B 0,C 180,E1 13086.206,E2 13086.206} C_VEL
LIN {X 0,Y 302.323,Z 751.811,A -85,B 0,C 180,E1 13082.709,E2 13082.709} C_VEL
LIN {X 0,Y 288.484,Z 727.615,A -85,B 0,C 180,E1 13079.059,E2 13079.059} C_VEL
LIN {X 0,Y 276.188,Z 707.258,A -85,B 0,C 180,E1 13075.465,E2 13075.465} C_VEL
LIN {X 0,Y 266.741,Z 692.711,A -85,B 0,C 180,E1 13072.482,E2 13072.482} C_VEL
LIN {X 0,Y 260.951,Z 684.024,A -85,B 0,C 180,E1 13070.527,E2 13070.527} C_VEL
LIN {X 0,Y 257.864,Z 679.38,A -85,B 0,C 180,E1 13069.424,E2 13069.424} C_VEL
LIN {X 0,Y 255.413,Z 675.39,A -85,B 0,C 180,E1 13068.49,E2 13068.49} C_VEL
LIN {X 0,Y 252.456,Z 671.598,A -85,B 0,C 180,E1 13067.414,E2 13067.414} C_VEL
LIN {X 0,Y 251.799,Z 669.292,A -85,B 0,C 180,E1 13067.026,E2 13067.026} C_VEL
LIN {X 0,Y 251.82,Z 669.289,A -85,B 0,C 180,E1 13062.151,E2 13062.151} C_VEL
LIN {X 0,Y 251.818,Z 669.287,A -85,B 0,C 180,E1 13057.074,E2 13057.074} C_VEL
LIN {X 0,Y 251.762,Z 669.283,A -85,B 0,C 180,E1 13051.824,E2 13051.824} C_VEL
LIN {X 0,Y 251.815,Z 669.274,A -85,B 0,C 180,E1 13047.044,E2 13047.044} C_VEL
LIN {X 0,Y 251.821,Z 669.299,A -85,B 0,C 180,E1 13042.015,E2 13042.015} C_VEL
LIN {X 0,Y 251.779,Z 669.283,A -85,B 0,C 180,E1 13036.92,E2 13036.92} C_VEL
LIN {X 0,Y 251.793,Z 669.301,A -85,B 0,C 180,E1 13031.96,E2 13031.96} C_VEL
LIN {X 0,Y 251.833,Z 669.295,A -85,B 0,C 180,E1 13027.078,E2 13027.078} C_VEL
LIN {X 0,Y 251.834,Z 669.39,A -85,B 0,C 180,E1 13023.728,E2 13023.728} C_VEL
LIN {X 0,Y 260.026,Z 691.522,A -85,B 0,C 180,E1 13019.501,E2 13019.501} C_VEL
LIN {X 0,Y 266.961,Z 711.966,A -85,B 0,C 180,E1 13015.952,E2 13015.952} C_VEL
LIN {X 0,Y 273.251,Z 733.453,A -85,B 0,C 180,E1 13012.468,E2 13012.468} C_VEL
LIN {X 0,Y 275.736,Z 742.981,A -85,B 0,C 180,E1 13011.017,E2 13011.017} C_VEL
LIN {X 0,Y 271.027,Z 786.491,A -85,B 0,C 180,E1 13005.998,E2 13005.998} C_VEL
LIN {X 0,Y 266.58,Z 830.555,A -85,B 0,C 180,E1 13000.876,E2 13000.876} C_VEL
LIN {X 0,Y 264.131,Z 854.54,A -85,B 0,C 180,E1 12998.094,E2 12998.094} C_VEL
